# B&R Automation Studio project CarWashSimu
Automation Studio 4.12.4.107 SP; technology packages: mapp 5.23.1, mappView 5.23.0

## Configuration Config1

CPU X20CP0484-1, AutomationRuntime B4.91, Build 4.1.2, Vc V4.72.9

### Task classes (Cpu.sw)
```
Cyclic#1 (cycle 2000 us, tolerance 2000 us):
  ComTCP_P <- Libraries.ComTCP.ComTCP_P.prg
  MainCtrl <- Source.MainCtrl.MainCtrl.prg
  EntryCtrl <- Source.Entrance.EntryCtrl.prg
  ChemCtrl <- Source.Chemicals.ChemCtrl.prg
  HPWater <- Source.HPWater.HPWater.prg
  HBrushCtrl <- Source.HBrush.HBrushCtrl.prg
  VBrushCtrl <- Source.VBrush.VBrushCtrl.prg
  UBCtrl <- Source.OptUnderBody.UBCtrl.prg
  HPolish <- Source.HPolishp.HPolish.prg
  VPolishCtr <- Source.OptVpolish.VPolishCtr.prg
  WaxCtrl <- Source.OptWax.WaxCtrl.prg
  DryHCtrl <- Source.Drying.DryHCtrl.prg
  DryH2Ctrl <- Source.Drying.DryH2Ctrl.prg
  CarExit <- Source.CarExit.CarExit.prg
  Auxillary <- Source.Auxillary.Auxillary.prg
Cyclic#3 (cycle 50000 us, tolerance 50000 us):
  AlarmCtrl <- Source.Infrastructure.AlarmCtrl.AlarmCtrl.prg
  RecipeCtrl <- Source.Infrastructure.RecipeCtrl.RecipeCtrl.prg
  DataCtrl <- Source.Infrastructure.DataCtrl.DataCtrl.prg
Cyclic#4 (cycle 100000 us, tolerance 100000 us):
  Dist <- Source.Dist.prg
Cyclic#5 (cycle 200000 us, tolerance 200000 us):
  VisuCtrl <- Source.VisuCtrl.VisuCtrl.prg
Binaries: FWRules, mvLoader, TCData, udbdef, iomap, asfw, Role, sysconf, arconfig, ashwd, User, ashwac
Libraries: ComTCP_L, AsTCP, operator, runtime, astime, standard, ArEventLog, AsBrStr, MpAlarmX, MpBase, MpData, FileIO, DataObj, sys_lib, brsystem, sys_lib, arssl, fileio, asieccon, brsystem, loopconr
```

### Hardware
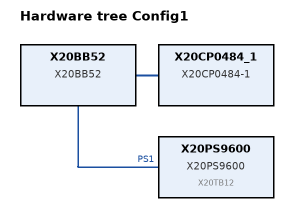
```
X20BB52 : X20BB52 v1.2.0.0
X20CP0484_1 : X20CP0484-1 v1.4.0.0  [SL -> X20BB52.SL1]
  Connector IF2:
    ActivateDevice = 1
  ConfigurationID = CarWashSimu_Config1
  Simulation = 1
  TimerDeviceType = SWIOTIMER
  Cyclic1Duration = 2000
  Cyclic1Tolerance = 2000
  Cyclic2Duration = 20000
  Cyclic2Tolerance = 20000
  Cyclic3Duration = 50000
  Cyclic3Tolerance = 50000
  Cyclic4Duration = 100000
  Cyclic4Tolerance = 100000
  Cyclic5Duration = 200000
  Cyclic5Tolerance = 200000
  Cyclic6Duration = 500000
  Cyclic6Tolerance = 500000
  Cyclic7Duration = 1000000
  Cyclic7Tolerance = 1000000
  Cyclic8Duration = 10000
  Cyclic8Tolerance = 30000000
  FileDevice1
  FileDeviceName1 = USER
  FileDevicePath1 = USER_PATH
X20PS9600 : X20PS9600 v1.6.0.0  [PS -> X20BB52.PS1; SS1 -> X20TB12.SS]
X20TB12 : X20TB12 v1.0.0.0
```

### PvMap.vvm - X20CP0484_1/PvMap.vvm
```iecst
VAR_CONFIG
	::ChemCtrl:iChem.IO.doChemRefill AT %Q.::ComTCP_SimOutputs.doChemRefill; (*Insert your comment here...*)
	::VPolishCtr:iVPolish.IO.aoVPLVel AT %Q.::ComTCP_SimOutputs.aoVPolishLVel; (*Insert your comment here...*)
	::VPolishCtr:iVPolish.IO.aoVPRVel AT %Q.::ComTCP_SimOutputs.aoVPolishRVel; (*Insert your comment here...*)
	::VPolishCtr:iVPolish.IO.doRelayRClose AT %Q.::ComTCP_SimOutputs.doVPolishRelayRClose; (*Insert your comment here...*)
	::VPolishCtr:iVPolish.IO.doRelayLClose AT %Q.::ComTCP_SimOutputs.doVPolishRelayLClose; (*Insert your comment here...*)
	::VPolishCtr:iVPolish.IO.doRelayLOpen AT %Q.::ComTCP_SimOutputs.doVPolishRelayLOpen; (*Insert your comment here...*)
	::VPolishCtr:iVPolish.IO.doRelayBrush AT %Q.::ComTCP_SimOutputs.doVPolishRelayBrush; (*Insert your comment here...*)
	::VPolishCtr:iVPolish.IO.doRelayROpen AT %Q.::ComTCP_SimOutputs.doVPolishRelayROpen; (*Insert your comment here...*)
	::ComTCP_SimInputs.aiVPolishRForceS AT %Q.::VPolishCtr:iVPolish.IO.aiVPRForceS; (*Insert your comment here...*)
	::ComTCP_SimInputs.aiVPolishRForceF AT %Q.::VPolishCtr:iVPolish.IO.aiVPRForceF; (*Insert your comment here...*)
	::ComTCP_SimInputs.aiVPolishLForceS AT %Q.::VPolishCtr:iVPolish.IO.aiVPLForceS; (*Insert your comment here...*)
	::ComTCP_SimInputs.aiVPolishLForceF AT %Q.::VPolishCtr:iVPolish.IO.aiVPLForceF; (*Insert your comment here...*)
	::CarExit:iExit.IO.doOrangeLight AT %Q.::ComTCP_SimOutputs.doExitOrangeLight; (*Insert your comment here...*)
	::CarExit:iExit.IO.doRedLight AT %Q.::ComTCP_SimOutputs.doExitRedLight; (*Insert your comment here...*)
	::ComTCP_SimOutputs.doExitGreenLight AT %Q.::ComTCP_SimOutputs.doExitGreenLight; (*Insert your comment here...*)
	::ComTCP_SimOutputs.doExitLiftDoorRelay AT %Q.::CarExit:iExit.IO.doRelayLiftDoor; (*Insert your comment here...*)
	::CarExit:iExit.IO.doRelayLowerdDoor AT %Q.::ComTCP_SimOutputs.doExitLowerDoorRelay; (*Insert your comment here...*)
	::MainCtrl:ScalDirt.y AT %Q.::ChemCtrl:iChem.IO.aoChemChemValve; (*Insert your comment here...*)
	::VBrushCtrl:iVBrush.Par.LeftVel AT %Q.::ComTCP_SimOutputs.aoVBrushLVel; (*Insert your comment here...*)
	::VBrushCtrl:iVBrush.Par.RightVel AT %Q.::ComTCP_SimOutputs.aoVBrushRVel; (*Insert your comment here...*)
	::Auxillary:iAuxillary.doRelayConv AT %Q.::ComTCP_SimOutputs.doConvRelay; (*Insert your comment here...*)
	::ChemCtrl:iChem.IO.doChemWaterValve AT %Q.::ComTCP_SimOutputs.doChemWaterValve; (*Insert your comment here...*)
	::ComTCP_SimInputs.aiEntranceSoilLevel AT %Q.::EntryCtrl:iEntry.IO.diSensSoilLvl; (*Insert your comment here...*)
	::ComTCP_SimInputs.aiVBrushLForceF AT %Q.::VBrushCtrl:iVBrush.IO.aiVBLForceF; (*Insert your comment here...*)
	::ComTCP_SimInputs.aiVBrushLForceS AT %Q.::VBrushCtrl:iVBrush.IO.aiVBLForceS; (*Insert your comment here...*)
	::ComTCP_SimInputs.aiVBrushRForceF AT %Q.::VBrushCtrl:iVBrush.IO.aiVBRForceF; (*Insert your comment here...*)
	::ComTCP_SimInputs.aiVBrushRForceS AT %Q.::VBrushCtrl:iVBrush.IO.aiVBRForceS; (*Insert your comment here...*)
	::ComTCP_SimInputs.diEmergencyStop AT %Q.::gMain.Cmd.EStop; (*Insert your comment here...*)
	::ComTCP_SimInputs.diEntranceSensor AT %Q.::EntryCtrl:iEntry.IO.diSensEntry; (*Insert your comment here...*)
	::ComTCP_SimInputs.diHBrushSensor1 AT %Q.::HBrushCtrl:iHBrush.IO.diSensHB1; (*Insert your comment here...*)
	::ComTCP_SimInputs.diHBrushSensor2 AT %Q.::HBrushCtrl:iHBrush.IO.diSensHB2; (*Insert your comment here...*)
	::ComTCP_SimInputs.diHBrushSensor3 AT %Q.::HBrushCtrl:iHBrush.IO.diSensHB3; (*Insert your comment here...*)
	::ComTCP_SimInputs.diHBrushSensor4 AT %Q.::HBrushCtrl:iHBrush.IO.diSensHB4; (*Insert your comment here...*)
	::ComTCP_SimInputs.diHighPressSensor1 AT %Q.::HPWater:iHighPress.IO.diSensHP1; (*Insert your comment here...*)
	::ComTCP_SimInputs.diHighPressSensor2 AT %Q.::HPWater:iHighPress.IO.diSensHP2; (*Insert your comment here...*)
	::ComTCP_SimInputs.diHighPressSensor3 AT %Q.::HPWater:iHighPress.IO.diSensHP3; (*Insert your comment here...*)
	::ComTCP_SimInputs.diHighPressSensor4 AT %Q.::HPWater:iHighPress.IO.diSensHP4; (*Insert your comment here...*)
	::ComTCP_SimInputs.diHPolishSensor1 AT %Q.::HPolish:iHPolish.IO.diSensHPolish1; (*Insert your comment here...*)
	::ComTCP_SimInputs.diHPolishSensor2 AT %Q.::HPolish:iHPolish.IO.diSensHPolish2; (*Insert your comment here...*)
	::ComTCP_SimInputs.diHPolishSensor3 AT %Q.::HPolish:iHPolish.IO.diSensHPolish3; (*Insert your comment here...*)
	::ComTCP_SimInputs.diHPolishSensor4 AT %Q.::HPolish:iHPolish.IO.diSensHPolish4; (*Insert your comment here...*)
	::HBrushCtrl:iHBrush.IO.doRelayHBBrush AT %Q.::ComTCP_SimOutputs.doHBrushBrushRelay; (*Insert your comment here...*)
	::HBrushCtrl:iHBrush.IO.doRelayHBLift AT %Q.::ComTCP_SimOutputs.doHBrushLiftRelay; (*Insert your comment here...*)
	::HBrushCtrl:iHBrush.IO.doRelayHBLower AT %Q.::ComTCP_SimOutputs.doHBrushLowerRelay; (*Insert your comment here...*)
	::HBrushCtrl:iHBrush.IO.doValveHB AT %Q.::ComTCP_SimOutputs.doHBrushValve; (*Insert your comment here...*)
	::HPolish:iHPolish.IO.doRelayBrush AT %Q.::ComTCP_SimOutputs.doHPolishBrushRelay; (*Insert your comment here...*)
	::HPolish:iHPolish.IO.doRelayLift AT %Q.::ComTCP_SimOutputs.doHPolishLiftRelay; (*Insert your comment here...*)
	::HPolish:iHPolish.IO.doRelayLower AT %Q.::ComTCP_SimOutputs.doHPolishLowerRelay; (*Insert your comment here...*)
	::HPWater:iHighPress.IO.doRelayHPLift AT %Q.::ComTCP_SimOutputs.doHighPressLiftRelay; (*Insert your comment here...*)
	::HPWater:iHighPress.IO.doRelayHPLow AT %Q.::ComTCP_SimOutputs.doHighPressLowerRelay; (*Insert your comment here...*)
	::HPWater:iHighPress.IO.doRelayHPPump AT %Q.::ComTCP_SimOutputs.doHighPressPumpRelay; (*Insert your comment here...*)
	::HPWater:iHighPress.IO.doValveHP AT %Q.::ComTCP_SimOutputs.doHighPressValve; (*Insert your comment here...*)
	::UBCtrl:iUBody.IO.doRelayPump AT %Q.::ComTCP_SimOutputs.doUnderbodyPumpRelay; (*Insert your comment here...*)
	::UBCtrl:iUBody.IO.doValveUB AT %Q.::ComTCP_SimOutputs.doUnderbodyValve; (*Insert your comment here...*)
	::VBrushCtrl:iVBrush.IO.doRelayVBLClose AT %Q.::ComTCP_SimOutputs.doVBrushRelayLClose; (*Insert your comment here...*)
	::VBrushCtrl:iVBrush.IO.doRelayVBLOpen AT %Q.::ComTCP_SimOutputs.doVBrushRelayLOpen; (*Insert your comment here...*)
	::VBrushCtrl:iVBrush.IO.doRelayVBRClose AT %Q.::ComTCP_SimOutputs.doVBrushRelayRClose; (*Insert your comment here...*)
	::VBrushCtrl:iVBrush.IO.doRelayVBROpen AT %Q.::ComTCP_SimOutputs.doVBrushRelayROpen; (*Insert your comment here...*)
	::ComTCP_SimInputs.diHDry1Sensor1 AT %Q.::DryHCtrl:iDry.IO.diSens1Dry1; (*Insert your comment here...*)
	::ComTCP_SimInputs.diHDry1Sensor2 AT %Q.::DryHCtrl:iDry.IO.diSens1Dry2; (*Insert your comment here...*)
	::ComTCP_SimInputs.diHDry1Sensor3 AT %Q.::DryHCtrl:iDry.IO.diSens1Dry3; (*Insert your comment here...*)
	::ComTCP_SimInputs.diHDry1Sensor4 AT %Q.::DryHCtrl:iDry.IO.diSens1Dry4; (*Insert your comment here...*)
	::ComTCP_SimInputs.diHDry2Sensor1 AT %Q.::DryH2Ctrl:iDry2.IO.diSens2Dry1; (*Insert your comment here...*)
	::ComTCP_SimInputs.diHDry2Sensor2 AT %Q.::DryH2Ctrl:iDry2.IO.diSens2Dry2; (*Insert your comment here...*)
	::ComTCP_SimInputs.diHDry2Sensor3 AT %Q.::DryH2Ctrl:iDry2.IO.diSens2Dry3; (*Insert your comment here...*)
	::ComTCP_SimInputs.diHDry2Sensor4 AT %Q.::DryH2Ctrl:iDry2.IO.diSens2Dry4; (*Insert your comment here...*)
	::DryHCtrl:iDry.IO.doRelayHD1Vent AT %Q.::ComTCP_SimOutputs.doHDry1VentRelay; (*Insert your comment here...*)
	::DryHCtrl:iDry.IO.doRelayHD1Heater AT %Q.::ComTCP_SimOutputs.doHDry1HeaterRelay; (*Insert your comment here...*)
	::DryHCtrl:iDry.IO.doRelayHD1Lower AT %Q.::ComTCP_SimOutputs.doHDry1LowerRelay; (*Insert your comment here...*)
	::DryHCtrl:iDry.IO.doRelayHD1Lift AT %Q.::ComTCP_SimOutputs.doHDry1LiftRelay; (*Insert your comment here...*)
	::DryH2Ctrl:iDry2.IO.doRelayHD2Vent AT %Q.::ComTCP_SimOutputs.doHDry2VentRelay; (*Insert your comment here...*)
	::DryH2Ctrl:iDry2.IO.doRelayHD2Heater AT %Q.::ComTCP_SimOutputs.doHDry2HeaterRelay; (*Insert your comment here...*)
	::DryH2Ctrl:iDry2.IO.doRelayHD2Lower AT %Q.::ComTCP_SimOutputs.doHDry2LowerRelay; (*Insert your comment here...*)
	::DryHCtrl:iDry.IO.doRelayVDHeater AT %Q.::ComTCP_SimOutputs.doVDry1HeaterRelay; (*Insert your comment here...*)
	::DryHCtrl:iDry.IO.doRelayVDVent AT %Q.::ComTCP_SimOutputs.doVDry1VentRelay; (*Insert your comment here...*)
	::DryH2Ctrl:iDry2.IO.doRelayHD2Lift AT %Q.::ComTCP_SimOutputs.doHDry2LiftRelay; (*Insert your comment here...*)
	::WaxCtrl:iWax.IO.doValveWax AT %Q.::ComTCP_SimOutputs.doWaxValve; (*Insert your comment here...*)
	::WaxCtrl:iWax.IO.doRefillWax AT %Q.::ComTCP_SimOutputs.doWaxRefill; (*Insert your comment here...*)
	::WaxCtrl:iWax.IO.doRealyWaxPump AT %Q.::ComTCP_SimOutputs.doWaxPumpRelay; (*Insert your comment here...*)
END_VAR
```

### Config.mpalarmxcore - X20CP0484_1/mappServices/Config.mpalarmxcore
```
Element gAlarmXCore (Type=mpalarmxcore)
  mapp.AlarmX.Core:
    BySeverity:
      [0]:
        Severity = 100
        [0] = Reaction
          Name = EStopErr
  mapp.AlarmX.Core.Configuration:
    [0]:
      Name = EStopChem
      Message = EStop Pressed chemical control
      Severity = 100
      Behavior = PersistentAlarm
    [1]:
      Name = EStopHighPre
      Message = EStop Pressed High pressurecontrol
      Severity = 100
      Behavior = PersistentAlarm
    [2]:
      Name = EStopHB
      Message = EStop Pressed horizontal brush control
      Severity = 100
      Behavior = PersistentAlarm
    [3]:
      Name = EStopVB
      Message = EStop Pressed vertical brush control
      Severity = 100
      Behavior = PersistentAlarm
    [4]:
      Name = EStopUB
      Message = EStop Pressed under body control
      Severity = 100
      Behavior = PersistentAlarm
    [5]:
      Name = EStopVPol
      Message = Estop Pressed Vertical polish
      Severity = 100
      Behavior = PersistentAlarm
    [6]:
      Name = EStopDry
      Message = EStop Pressed Dry control
      Severity = 100
      Behavior = PersistentAlarm
    [7]:
      Name = EStopHWax
      Message = EStop Pressed HotWax control
      Severity = 100
      Behavior = PersistentAlarm
    [8]:
      Name = EStopConv
      Message = EStop Pressed Conveyor control
      Severity = 100
      Behavior = PersistentAlarm
    [9]:
      Name = WaterLow
      Message = Water level is low
      Severity = 100
      Behavior = PersistentAlarm
    [10]:
      Name = ChemLow
      Message = Chemical level is low
      Severity = 50
      Behavior = PersistentAlarm
    [11]:
      Name = WaxLow
      Message = Wax level is low
      Severity = 50
      Behavior = PersistentAlarm
    [12]:
      Name = EStopEntry
      Message = Emergency stop of entry is pressed
      Severity = 100
      Behavior = PersistentAlarm
    [13]:
      Name = EStopHPol
      Message = Estop Pressed Horizonatal polish
      Severity = 100
      Behavior = PersistentAlarm
    [14]:
      Name = EStopExit
      Message = EStop of exit is pressed
      Severity = 100
      Behavior = PersistentAlarm
Element gAlarmXCore_1 (Type=mpalarmxcore)
```

## Logical view

Binary libraries used (declarations not repeated): operator, runtime, astime, AsIecCon, AsTCP, standard, ArEventLog, AsBrStr, LoopConR, sys_lib, brsystem, MpAlarmX, MpBase, MpData, FileIO, DataObj

### Global.typ - Global data types
```iecst
TYPE
	MainCmd_typ : 	STRUCT
		Start : BOOL;
		Stop : BOOL;
		EStop : BOOL;
	END_STRUCT;
	MainOption_typ : 	STRUCT
		EntryState : BOOL;
		ChemicalState : BOOL;
		HighPress : BOOL;
		HBrush : BOOL;
		Polish : BOOL;
		UnderBody : BOOL;
		Wax : BOOL;
		VBrush : BOOL;
		Dry : BOOL;
	END_STRUCT;
	MainCtrl_typ : 	STRUCT
		Cmd : MainCmd_typ;
		Option : MainOption_typ;
	END_STRUCT;
END_TYPE
```

### Global.var - Global variables
```iecst
VAR
	gMi_Mode2 : BOOL;
	gMi_Mode3 : BOOL;
	gMi_Mode4 : BOOL;
	gMi_Mode1 : BOOL;
	gMain : MainCtrl_typ;
	iVa_Distance : REAL;
	gCar : ARRAY[0..2] OF BOOL;
END_VAR
```

### Package Logical/Libraries - Global libraries

### Library Logical/Libraries/ComTCP/ComTCP_L (ANSIC)
Depends on: AsTCP, operator, runtime, astime, standard, ArEventLog, AsBrStr

#### MNG_Global.hpp
```cpp
#ifndef  _MNGGLOBAL_HPP_
#define _MNGGLOBAL_HPP_

#include <mng_globalTYP.h>

    typedef struct {

		signed short NumSignals;

        /* BOOL diEmergencyStop */
        BOOL diEmergencyStop;
        /* BOOL diEntranceSensor */
        BOOL diEntranceSensor;
        /* REAL aiEntranceSoilLevel */
        REAL aiEntranceSoilLevel;
        /* BOOL diHighPressSensor1 */
        BOOL diHighPressSensor1;
        /* BOOL diHighPressSensor2 */
        BOOL diHighPressSensor2;
        /* BOOL diHighPressSensor3 */
        BOOL diHighPressSensor3;
        /* BOOL diHighPressSensor4 */
        BOOL diHighPressSensor4;
        /* BOOL diHBrushSensor1 */
        BOOL diHBrushSensor1;
        /* BOOL diHBrushSensor2 */
        BOOL diHBrushSensor2;
        /* BOOL diHBrushSensor3 */
        BOOL diHBrushSensor3;
        /* BOOL diHBrushSensor4 */
        BOOL diHBrushSensor4;
        /* REAL aiVBrushLForceF */
        REAL aiVBrushLForceF;
        /* REAL aiVBrushLForceS */
        REAL aiVBrushLForceS;
        /* REAL aiVBrushRForceF */
        REAL aiVBrushRForceF;
        /* REAL aiVBrushRForceS */
        REAL aiVBrushRForceS;
        /* BOOL diHPolishSensor1 */
        BOOL diHPolishSensor1;
        /* BOOL diHPolishSensor2 */
        BOOL diHPolishSensor2;
        /* BOOL diHPolishSensor3 */
        BOOL diHPolishSensor3;
        /* BOOL diHPolishSensor4 */
        BOOL diHPolishSensor4;
        /* REAL aiVPolishLForceF */
        REAL aiVPolishLForceF;
        /* REAL aiVPolishLForceS */
        REAL aiVPolishLForceS;
        /* REAL aiVPolishRForceF */
        REAL aiVPolishRForceF;
        /* REAL aiVPolishRForceS */
        REAL aiVPolishRForceS;
        /* BOOL diHDry1Sensor1 */
        BOOL diHDry1Sensor1;
        /* BOOL diHDry1Sensor2 */
        BOOL diHDry1Sensor2;
        /* BOOL diHDry1Sensor3 */
        BOOL diHDry1Sensor3;
        /* BOOL diHDry1Sensor4 */
        BOOL diHDry1Sensor4;
        /* BOOL diHDry2Sensor1 */
        BOOL diHDry2Sensor1;
        /* BOOL diHDry2Sensor2 */
        BOOL diHDry2Sensor2;
        /* BOOL diHDry2Sensor3 */
        BOOL diHDry2Sensor3;
        /* BOOL diHDry2Sensor4 */
        BOOL diHDry2Sensor4;
        /* REAL aiWaterLevel */
        REAL aiWaterLevel;

        } ComTCP_INPUTS_32BIT_FWRD;

    typedef struct {

		signed short NumSignals;

        /* BOOL doMaintenanceMode */
        BOOL doMaintenanceMode;
        /* REAL aoChemChemValve */
        REAL aoChemChemValve;
        /* BOOL doChemWaterValve */
        BOOL doChemWaterValve;
        /* BOOL doChemRefill */
        BOOL doChemRefill;
        /* BOOL doHighPressLiftRelay */
        BOOL doHighPressLiftRelay;
        /* BOOL doHighPressLowerRelay */
        BOOL doHighPressLowerRelay;
        /* BOOL doHighPressValve */
        BOOL doHighPressValve;
        /* BOOL doHighPressPumpRelay */
        BOOL doHighPressPumpRelay;
        /* BOOL doHBrushLiftRelay */
        BOOL doHBrushLiftRelay;
        /* BOOL doHBrushLowerRelay */
        BOOL doHBrushLowerRelay;
        /* BOOL doHBrushValve */
        BOOL doHBrushValve;
        /* BOOL doHBrushBrushRelay */
        BOOL doHBrushBrushRelay;
        /* BOOL doVBrushRelayLClose */
        BOOL doVBrushRelayLClose;
        /* BOOL doVBrushRelayLOpen */
        BOOL doVBrushRelayLOpen;
        /* BOOL doVBrushRelayRClose */
        BOOL doVBrushRelayRClose;
        /* BOOL doVBrushRelayROpen */
        BOOL doVBrushRelayROpen;
        /* REAL aoVBrushLVel */
        REAL aoVBrushLVel;
        /* REAL aoVBrushRVel */
        REAL aoVBrushRVel;
        /* BOOL doVBrushValve */
        BOOL doVBrushValve;
        /* BOOL doVBrushRelayBrush */
        BOOL doVBrushRelayBrush;
        /* BOOL doUnderbodyValve */
        BOOL doUnderbodyValve;
        /* BOOL doUnderbodyPumpRelay */
        BOOL doUnderbodyPumpRelay;
        /* BOOL doHPolishLiftRelay */
        BOOL doHPolishLiftRelay;
        /* BOOL doHPolishLowerRelay */
        BOOL doHPolishLowerRelay;
        /* BOOL doHPolishBrushRelay */
        BOOL doHPolishBrushRelay;
        /* BOOL doVPolishRelayLClose */
        BOOL doVPolishRelayLClose;
        /* BOOL doVPolishRelayLOpen */
        BOOL doVPolishRelayLOpen;
        /* BOOL doVPolishRelayRClose */
        BOOL doVPolishRelayRClose;
        /* BOOL doVPolishRelayROpen */
        BOOL doVPolishRelayROpen;
        /* REAL aoVPolishLVel */
        REAL aoVPolishLVel;
        /* REAL aoVPolishRVel */
        REAL aoVPolishRVel;
        /* BOOL doVPolishRelayBrush */
        BOOL doVPolishRelayBrush;
        /* BOOL doWaxValve */
        BOOL doWaxValve;
        /* BOOL doWaxPumpRelay */
        BOOL doWaxPumpRelay;
        /* BOOL doWaxRefill */
        BOOL doWaxRefill;
        /* BOOL doHDry1LiftRelay */
        BOOL doHDry1LiftRelay;
        /* BOOL doHDry1LowerRelay */
        BOOL doHDry1LowerRelay;
        /* BOOL doHDry1VentRelay */
        BOOL doHDry1VentRelay;
        /* BOOL doHDry1HeaterRelay */
        BOOL doHDry1HeaterRelay;
        /* BOOL doVDry1VentRelay */
        BOOL doVDry1VentRelay;
        /* BOOL doVDry1HeaterRelay */
        BOOL doVDry1HeaterRelay;
        /* BOOL doHDry2LiftRelay */
        BOOL doHDry2LiftRelay;
        /* BOOL doHDry2LowerRelay */
        BOOL doHDry2LowerRelay;
        /* BOOL doHDry2VentRelay */
        BOOL doHDry2VentRelay;
        /* BOOL doHDry2HeaterRelay */
        BOOL doHDry2HeaterRelay;
        /* BOOL doConvRelay */
        BOOL doConvRelay;
        /* BOOL doWaterValve */
        BOOL doWaterValve;
        /* BOOL doTankWaterValve */
        BOOL doTankWaterValve;
        /* BOOL doExitGreenLight */
        BOOL doExitGreenLight;
        /* BOOL doExitOrangeLight */
        BOOL doExitOrangeLight;
        /* BOOL doExitRedLight */
        BOOL doExitRedLight;
        /* BOOL doExitLiftDoorRelay */
        BOOL doExitLiftDoorRelay;
        /* BOOL doExitLowerDoorRelay */
        BOOL doExitLowerDoorRelay;

        } ComTCP_OUTPUTS_32BIT_FWRD;

#endif
```

#### MNG_CpyOutToMsg.cpp
```cpp
#include "MNG_InternalTyp.hpp"

unsigned long int MNG_CpyOutToMsg(MNG_RawDatagram * pToServer, unsigned long int counter, ComTCP_OUTPUTS_32BIT_FWRD *pSimOutputs ) {

        unsigned long int DWordBuffer;

        pSimOutputs->NumSignals = 53;
        (pToServer->Header).ByteCount    = H_TO_NUDINT(216);
        (pToServer->Header).DatagramType = H_TO_NUDINT(MNG_Raw32BitImage);
        (pToServer->Header).SentTime = H_TO_NUDINT(0);  // Todo
        (pToServer->Header).Counter = H_TO_NUDINT(counter);
        pToServer->Payload[0] = H_TO_NUDINT(pSimOutputs->NumSignals);

    /* doMaintenanceMode : BOOL */
    if(pSimOutputs->doMaintenanceMode == 1) {
        pToServer->Payload[1] = 0xFFFFFFFF;   /*BOOL */
    } else {
        pToServer->Payload[1] = 0;
    }

    /* aoChemChemValve : FLOAT32 */
    brsmemcpy((unsigned long int)&(DWordBuffer), (unsigned long int)&(pSimOutputs->aoChemChemValve), 4);
    pToServer->Payload[2] = H_TO_NUDINT(DWordBuffer);

    /* doChemWaterValve : BOOL */
    if(pSimOutputs->doChemWaterValve == 1) {
        pToServer->Payload[3] = 0xFFFFFFFF;   /*BOOL */
    } else {
        pToServer->Payload[3] = 0;
    }

    /* doChemRefill : BOOL */
    if(pSimOutputs->doChemRefill == 1) {
        pToServer->Payload[4] = 0xFFFFFFFF;   /*BOOL */
    } else {
        pToServer->Payload[4] = 0;
    }

    /* doHighPressLiftRelay : BOOL */
    if(pSimOutputs->doHighPressLiftRelay == 1) {
        pToServer->Payload[5] = 0xFFFFFFFF;   /*BOOL */
    } else {
        pToServer->Payload[5] = 0;
    }

    /* doHighPressLowerRelay : BOOL */
    if(pSimOutputs->doHighPressLowerRelay == 1) {
        pToServer->Payload[6] = 0xFFFFFFFF;   /*BOOL */
    } else {
        pToServer->Payload[6] = 0;
    }

    /* doHighPressValve : BOOL */
    if(pSimOutputs->doHighPressValve == 1) {
        pToServer->Payload[7] = 0xFFFFFFFF;   /*BOOL */
    } else {
        pToServer->Payload[7] = 0;
    }

    /* doHighPressPumpRelay : BOOL */
    if(pSimOutputs->doHighPressPumpRelay == 1) {
        pToServer->Payload[8] = 0xFFFFFFFF;   /*BOOL */
    } else {
        pToServer->Payload[8] = 0;
    }

    /* doHBrushLiftRelay : BOOL */
    if(pSimOutputs->doHBrushLiftRelay == 1) {
        pToServer->Payload[9] = 0xFFFFFFFF;   /*BOOL */
    } else {
        pToServer->Payload[9] = 0;
    }

    /* doHBrushLowerRelay : BOOL */
    if(pSimOutputs->doHBrushLowerRelay == 1) {
        pToServer->Payload[10] = 0xFFFFFFFF;   /*BOOL */
    } else {
        pToServer->Payload[10] = 0;
    }

    /* doHBrushValve : BOOL */
    if(pSimOutputs->doHBrushValve == 1) {
        pToServer->Payload[11] = 0xFFFFFFFF;   /*BOOL */
    } else {
        pToServer->Payload[11] = 0;
    }

    /* doHBrushBrushRelay : BOOL */
    if(pSimOutputs->doHBrushBrushRelay == 1) {
        pToServer->Payload[12] = 0xFFFFFFFF;   /*BOOL */
    } else {
        pToServer->Payload[12] = 0;
    }

    /* doVBrushRelayLClose : BOOL */
    if(pSimOutputs->doVBrushRelayLClose == 1) {
        pToServer->Payload[13] = 0xFFFFFFFF;   /*BOOL */
    } else {
        pToServer->Payload[13] = 0;
    }

    /* doVBrushRelayLOpen : BOOL */
    if(pSimOutputs->doVBrushRelayLOpen == 1) {
        pToServer->Payload[14] = 0xFFFFFFFF;   /*BOOL */
    } else {
        pToServer->Payload[14] = 0;
    }

    /* doVBrushRelayRClose : BOOL */
    if(pSimOutputs->doVBrushRelayRClose == 1) {
        pToServer->Payload[15] = 0xFFFFFFFF;   /*BOOL */
    } else {
        pToServer->Payload[15] = 0;
    }

    /* doVBrushRelayROpen : BOOL */
    if(pSimOutputs->doVBrushRelayROpen == 1) {
        pToServer->Payload[16] = 0xFFFFFFFF;   /*BOOL */
    } else {
        pToServer->Payload[16] = 0;
    }

    /* aoVBrushLVel : FLOAT32 */
    brsmemcpy((unsigned long int)&(DWordBuffer), (unsigned long int)&(pSimOutputs->aoVBrushLVel), 4);
    pToServer->Payload[17] = H_TO_NUDINT(DWordBuffer);

    /* aoVBrushRVel : FLOAT32 */
    brsmemcpy((unsigned long int)&(DWordBuffer), (unsigned long int)&(pSimOutputs->aoVBrushRVel), 4);
    pToServer->Payload[18] = H_TO_NUDINT(DWordBuffer);

    /* doVBrushValve : BOOL */
    if(pSimOutputs->doVBrushValve == 1) {
        pToServer->Payload[19] = 0xFFFFFFFF;   /*BOOL */
    } else {
        pToServer->Payload[19] = 0;
    }

    /* doVBrushRelayBrush : BOOL */
    if(pSimOutputs->doVBrushRelayBrush == 1) {
        pToServer->Payload[20] = 0xFFFFFFFF;   /*BOOL */
    } else {
        pToServer->Payload[20] = 0;
    }

    /* doUnderbodyValve : BOOL */
    if(pSimOutputs->doUnderbodyValve == 1) {
        pToServer->Payload[21] = 0xFFFFFFFF;   /*BOOL */
    } else {
        pToServer->Payload[21] = 0;
    }

    /* doUnderbodyPumpRelay : BOOL */
    if(pSimOutputs->doUnderbodyPumpRelay == 1) {
        pToServer->Payload[22] = 0xFFFFFFFF;   /*BOOL */
    } else {
        pToServer->Payload[22] = 0;
    }

    /* doHPolishLiftRelay : BOOL */
    if(pSimOutputs->doHPolishLiftRelay == 1) {
        pToServer->Payload[23] = 0xFFFFFFFF;   /*BOOL */
    } else {
        pToServer->Payload[23] = 0;
    }

    /* doHPolishLowerRelay : BOOL */
    if(pSimOutputs->doHPolishLowerRelay == 1) {
        pToServer->Payload[24] = 0xFFFFFFFF;   /*BOOL */
    } else {
        pToServer->Payload[24] = 0;
    }

    /* doHPolishBrushRelay : BOOL */
    if(pSimOutputs->doHPolishBrushRelay == 1) {
        pToServer->Payload[25] = 0xFFFFFFFF;   /*BOOL */
    } else {
        pToServer->Payload[25] = 0;
    }

    /* doVPolishRelayLClose : BOOL */
    if(pSimOutputs->doVPolishRelayLClose == 1) {
        pToServer->Payload[26] = 0xFFFFFFFF;   /*BOOL */
    } else {
        pToServer->Payload[26] = 0;
    }

    /* doVPolishRelayLOpen : BOOL */
    if(pSimOutputs->doVPolishRelayLOpen == 1) {
        pToServer->Payload[27] = 0xFFFFFFFF;   /*BOOL */
    } else {
        pToServer->Payload[27] = 0;
    }

    /* doVPolishRelayRClose : BOOL */
    if(pSimOutputs->doVPolishRelayRClose == 1) {
        pToServer->Payload[28] = 0xFFFFFFFF;   /*BOOL */
    } else {
        pToServer->Payload[28] = 0;
    }

    /* doVPolishRelayROpen : BOOL */
    if(pSimOutputs->doVPolishRelayROpen == 1) {
        pToServer->Payload[29] = 0xFFFFFFFF;   /*BOOL */
    } else {
        pToServer->Payload[29] = 0;
    }

    /* aoVPolishLVel : FLOAT32 */
    brsmemcpy((unsigned long int)&(DWordBuffer), (unsigned long int)&(pSimOutputs->aoVPolishLVel), 4);
    pToServer->Payload[30] = H_TO_NUDINT(DWordBuffer);

    /* aoVPolishRVel : FLOAT32 */
    brsmemcpy((unsigned long int)&(DWordBuffer), (unsigned long int)&(pSimOutputs->aoVPolishRVel), 4);
    pToServer->Payload[31] = H_TO_NUDINT(DWordBuffer);

    /* doVPolishRelayBrush : BOOL */
    if(pSimOutputs->doVPolishRelayBrush == 1) {
        pToServer->Payload[32] = 0xFFFFFFFF;   /*BOOL */
    } else {
        pToServer->Payload[32] = 0;
    }

    /* doWaxValve : BOOL */
    if(pSimOutputs->doWaxValve == 1) {
        pToServer->Payload[33] = 0xFFFFFFFF;   /*BOOL */
    } else {
        pToServer->Payload[33] = 0;
    }

    /* doWaxPumpRelay : BOOL */
    if(pSimOutputs->doWaxPumpRelay == 1) {
        pToServer->Payload[34] = 0xFFFFFFFF;   /*BOOL */
    } else {
        pToServer->Payload[34] = 0;
    }

    /* doWaxRefill : BOOL */
    if(pSimOutputs->doWaxRefill == 1) {
        pToServer->Payload[35] = 0xFFFFFFFF;   /*BOOL */
    } else {
        pToServer->Payload[35] = 0;
    }

    /* doHDry1LiftRelay : BOOL */
    if(pSimOutputs->doHDry1LiftRelay == 1) {
        pToServer->Payload[36] = 0xFFFFFFFF;   /*BOOL */
    } else {
        pToServer->Payload[36] = 0;
    }

    /* doHDry1LowerRelay : BOOL */
    if(pSimOutputs->doHDry1LowerRelay == 1) {
        pToServer->Payload[37] = 0xFFFFFFFF;   /*BOOL */
    } else {
        pToServer->Payload[37] = 0;
    }

    /* doHDry1VentRelay : BOOL */
    if(pSimOutputs->doHDry1VentRelay == 1) {
        pToServer->Payload[38] = 0xFFFFFFFF;   /*BOOL */
    } else {
        pToServer->Payload[38] = 0;
    }

    /* doHDry1HeaterRelay : BOOL */
    if(pSimOutputs->doHDry1HeaterRelay == 1) {
        pToServer->Payload[39] = 0xFFFFFFFF;   /*BOOL */
    } else {
        pToServer->Payload[39] = 0;
    }

    /* doVDry1VentRelay : BOOL */
    if(pSimOutputs->doVDry1VentRelay == 1) {
        pToServer->Payload[40] = 0xFFFFFFFF;   /*BOOL */
    } else {
        pToServer->Payload[40] = 0;
    }

    /* doVDry1HeaterRelay : BOOL */
    if(pSimOutputs->doVDry1HeaterRelay == 1) {
        pToServer->Payload[41] = 0xFFFFFFFF;   /*BOOL */
    } else {
        pToServer->Payload[41] = 0;
    }

    /* doHDry2LiftRelay : BOOL */
    if(pSimOutputs->doHDry2LiftRelay == 1) {
        pToServer->Payload[42] = 0xFFFFFFFF;   /*BOOL */
    } else {
        pToServer->Payload[42] = 0;
    }

    /* doHDry2LowerRelay : BOOL */
    if(pSimOutputs->doHDry2LowerRelay == 1) {
        pToServer->Payload[43] = 0xFFFFFFFF;   /*BOOL */
    } else {
        pToServer->Payload[43] = 0;
    }

    /* doHDry2VentRelay : BOOL */
    if(pSimOutputs->doHDry2VentRelay == 1) {
        pToServer->Payload[44] = 0xFFFFFFFF;   /*BOOL */
    } else {
        pToServer->Payload[44] = 0;
    }

    /* doHDry2HeaterRelay : BOOL */
    if(pSimOutputs->doHDry2HeaterRelay == 1) {
        pToServer->Payload[45] = 0xFFFFFFFF;   /*BOOL */
    } else {
        pToServer->Payload[45] = 0;
    }

    /* doConvRelay : BOOL */
    if(pSimOutputs->doConvRelay == 1) {
        pToServer->Payload[46] = 0xFFFFFFFF;   /*BOOL */
    } else {
        pToServer->Payload[46] = 0;
    }

    /* doWaterValve : BOOL */
    if(pSimOutputs->doWaterValve == 1) {
        pToServer->Payload[47] = 0xFFFFFFFF;   /*BOOL */
    } else {
        pToServer->Payload[47] = 0;
    }

    /* doTankWaterValve : BOOL */
    if(pSimOutputs->doTankWaterValve == 1) {
        pToServer->Payload[48] = 0xFFFFFFFF;   /*BOOL */
    } else {
        pToServer->Payload[48] = 0;
    }

    /* doExitGreenLight : BOOL */
    if(pSimOutputs->doExitGreenLight == 1) {
        pToServer->Payload[49] = 0xFFFFFFFF;   /*BOOL */
    } else {
        pToServer->Payload[49] = 0;
    }

    /* doExitOrangeLight : BOOL */
    if(pSimOutputs->doExitOrangeLight == 1) {
        pToServer->Payload[50] = 0xFFFFFFFF;   /*BOOL */
    } else {
        pToServer->Payload[50] = 0;
    }

    /* doExitRedLight : BOOL */
    if(pSimOutputs->doExitRedLight == 1) {
        pToServer->Payload[51] = 0xFFFFFFFF;   /*BOOL */
    } else {
        pToServer->Payload[51] = 0;
    }

    /* doExitLiftDoorRelay : BOOL */
    if(pSimOutputs->doExitLiftDoorRelay == 1) {
        pToServer->Payload[52] = 0xFFFFFFFF;   /*BOOL */
    } else {
        pToServer->Payload[52] = 0;
    }

    /* doExitLowerDoorRelay : BOOL */
    if(pSimOutputs->doExitLowerDoorRelay == 1) {
        pToServer->Payload[53] = 0xFFFFFFFF;   /*BOOL */
    } else {
        pToServer->Payload[53] = 0;
    }

	return 0;
}
```

#### MNG_CpyMsgToInp.cpp
```cpp
#include "MNG_InternalTyp.hpp"

unsigned long int MNG_CpyMsgToInp(MNG_RawDatagram * pFromServer, ComTCP_INPUTS_32BIT_FWRD *pSimInputs) {

    MNG_DatagramType datagramType;
	unsigned long int DWordBuffer;
        unsigned long int byteCount;
	unsigned long int numSignalsInMessage;

	byteCount = N_TO_HUDINT((pFromServer->Header).ByteCount);
	datagramType = static_cast<MNG_DatagramType>(N_TO_HUDINT((pFromServer->Header).DatagramType));
	if (datagramType != MNG_Raw32BitImage) {
		return 0;
	}

    pSimInputs->NumSignals = 32;

    numSignalsInMessage = N_TO_HUDINT(pFromServer->Payload[0]);
        if ((static_cast<long int>(numSignalsInMessage) != pSimInputs->NumSignals) ||
	(byteCount != 4 + numSignalsInMessage * 4)) {
		return 0;
	}

    /* BOOL diEmergencyStop */
    pSimInputs->diEmergencyStop = (pFromServer->Payload[1] != 0);

    /* BOOL diEntranceSensor */
    pSimInputs->diEntranceSensor = (pFromServer->Payload[2] != 0);

    /* FLOAT32 aiEntranceSoilLevel */
    DWordBuffer = N_TO_HUDINT(pFromServer->Payload[3]);
    brsmemcpy((unsigned long int)&(pSimInputs->aiEntranceSoilLevel), (unsigned long int)&(DWordBuffer), 4);

    /* BOOL diHighPressSensor1 */
    pSimInputs->diHighPressSensor1 = (pFromServer->Payload[4] != 0);

    /* BOOL diHighPressSensor2 */
    pSimInputs->diHighPressSensor2 = (pFromServer->Payload[5] != 0);

    /* BOOL diHighPressSensor3 */
    pSimInputs->diHighPressSensor3 = (pFromServer->Payload[6] != 0);

    /* BOOL diHighPressSensor4 */
    pSimInputs->diHighPressSensor4 = (pFromServer->Payload[7] != 0);

    /* BOOL diHBrushSensor1 */
    pSimInputs->diHBrushSensor1 = (pFromServer->Payload[8] != 0);

    /* BOOL diHBrushSensor2 */
    pSimInputs->diHBrushSensor2 = (pFromServer->Payload[9] != 0);

    /* BOOL diHBrushSensor3 */
    pSimInputs->diHBrushSensor3 = (pFromServer->Payload[10] != 0);

    /* BOOL diHBrushSensor4 */
    pSimInputs->diHBrushSensor4 = (pFromServer->Payload[11] != 0);

    /* FLOAT32 aiVBrushLForceF */
    DWordBuffer = N_TO_HUDINT(pFromServer->Payload[12]);
    brsmemcpy((unsigned long int)&(pSimInputs->aiVBrushLForceF), (unsigned long int)&(DWordBuffer), 4);

    /* FLOAT32 aiVBrushLForceS */
    DWordBuffer = N_TO_HUDINT(pFromServer->Payload[13]);
    brsmemcpy((unsigned long int)&(pSimInputs->aiVBrushLForceS), (unsigned long int)&(DWordBuffer), 4);

    /* FLOAT32 aiVBrushRForceF */
    DWordBuffer = N_TO_HUDINT(pFromServer->Payload[14]);
    brsmemcpy((unsigned long int)&(pSimInputs->aiVBrushRForceF), (unsigned long int)&(DWordBuffer), 4);

    /* FLOAT32 aiVBrushRForceS */
    DWordBuffer = N_TO_HUDINT(pFromServer->Payload[15]);
    brsmemcpy((unsigned long int)&(pSimInputs->aiVBrushRForceS), (unsigned long int)&(DWordBuffer), 4);

    /* BOOL diHPolishSensor1 */
    pSimInputs->diHPolishSensor1 = (pFromServer->Payload[16] != 0);

    /* BOOL diHPolishSensor2 */
    pSimInputs->diHPolishSensor2 = (pFromServer->Payload[17] != 0);

    /* BOOL diHPolishSensor3 */
    pSimInputs->diHPolishSensor3 = (pFromServer->Payload[18] != 0);

    /* BOOL diHPolishSensor4 */
    pSimInputs->diHPolishSensor4 = (pFromServer->Payload[19] != 0);

    /* FLOAT32 aiVPolishLForceF */
    DWordBuffer = N_TO_HUDINT(pFromServer->Payload[20]);
    brsmemcpy((unsigned long int)&(pSimInputs->aiVPolishLForceF), (unsigned long int)&(DWordBuffer), 4);

    /* FLOAT32 aiVPolishLForceS */
    DWordBuffer = N_TO_HUDINT(pFromServer->Payload[21]);
    brsmemcpy((unsigned long int)&(pSimInputs->aiVPolishLForceS), (unsigned long int)&(DWordBuffer), 4);

    /* FLOAT32 aiVPolishRForceF */
    DWordBuffer = N_TO_HUDINT(pFromServer->Payload[22]);
    brsmemcpy((unsigned long int)&(pSimInputs->aiVPolishRForceF), (unsigned long int)&(DWordBuffer), 4);

    /* FLOAT32 aiVPolishRForceS */
    DWordBuffer = N_TO_HUDINT(pFromServer->Payload[23]);
    brsmemcpy((unsigned long int)&(pSimInputs->aiVPolishRForceS), (unsigned long int)&(DWordBuffer), 4);

    /* BOOL diHDry1Sensor1 */
    pSimInputs->diHDry1Sensor1 = (pFromServer->Payload[24] != 0);

    /* BOOL diHDry1Sensor2 */
    pSimInputs->diHDry1Sensor2 = (pFromServer->Payload[25] != 0);

    /* BOOL diHDry1Sensor3 */
    pSimInputs->diHDry1Sensor3 = (pFromServer->Payload[26] != 0);

    /* BOOL diHDry1Sensor4 */
    pSimInputs->diHDry1Sensor4 = (pFromServer->Payload[27] != 0);

    /* BOOL diHDry2Sensor1 */
    pSimInputs->diHDry2Sensor1 = (pFromServer->Payload[28] != 0);

    /* BOOL diHDry2Sensor2 */
    pSimInputs->diHDry2Sensor2 = (pFromServer->Payload[29] != 0);

    /* BOOL diHDry2Sensor3 */
    pSimInputs->diHDry2Sensor3 = (pFromServer->Payload[30] != 0);

    /* BOOL diHDry2Sensor4 */
    pSimInputs->diHDry2Sensor4 = (pFromServer->Payload[31] != 0);

    /* FLOAT32 aiWaterLevel */
    DWordBuffer = N_TO_HUDINT(pFromServer->Payload[32]);
    brsmemcpy((unsigned long int)&(pSimInputs->aiWaterLevel), (unsigned long int)&(DWordBuffer), 4);

return N_TO_HUDINT((pFromServer->Header).Counter); // return counter
}
```

### Program Logical/Libraries/ComTCP/ComTCP_P (ANSIC)

#### Main.cpp
```cpp
#include <bur/plctypes.h>

#include "../ComTCP_L/MNG_Global.hpp"
#include "../ComTCP_L/MNG_InternalTyp.hpp"
#include "../ComTCP_L/MNG_ComHdlr.hpp"

#include <MNG_PackageTyp.h>
#include <MNG_PackageVAR.h>
#include <TypesTYP.h>
#include <VariablesVAR.h>

unsigned long bur_heap_size = 0x4FFFF;

MNG_ComHdlr *pMNG_ComHdlr;

void _INIT ProgramInit(void)
{
    pMNG_ComHdlr = new MNG_ComHdlr(ComTCP_SimServerAddress, ComTCP_SimServerPort, ComTCP_SimSendCycleTime);
}

void _CYCLIC ProgramCyclic(void)
{
    connectionState = pMNG_ComHdlr->RunCommunication((void*)&ComTCP_SimInputs,(void*)&ComTCP_SimOutputs, &ComTCP_SimActive);
}

void _EXIT ProgramExit(void)
{
    delete pMNG_ComHdlr;
}
```

### MNG_Package.typ
```iecst
(*                                                                            *)
(* File generated by the B&R AS 4 control config generator                    *)
(*                                                                            *)
(*     Provider: machineering                                                 *)
(*  Application: iPhysics_2.4.master                                          *)
(* Architecture: Windows 64 Bit                                               *)
(*      Version: 2.4.12706.master                                             *)
(*        Build: 608a88cb4                                                    *)
(*         Date: 2022-08-25, Time: 10:57:22                                   *)
(*                                                                            *)

TYPE
ComTCP_INPUTS_32BIT : STRUCT

		NumSignals	: INT := 32;

        diEmergencyStop : BOOL := 0;
        (* BOOL diEmergencyStop *)
        diEntranceSensor : BOOL := 0;
        (* BOOL diEntranceSensor *)
        aiEntranceSoilLevel : REAL := 0.0;
        (* REAL aiEntranceSoilLevel *)
        diHighPressSensor1 : BOOL := 0;
        (* BOOL diHighPressSensor1 *)
        diHighPressSensor2 : BOOL := 0;
        (* BOOL diHighPressSensor2 *)
        diHighPressSensor3 : BOOL := 0;
        (* BOOL diHighPressSensor3 *)
        diHighPressSensor4 : BOOL := 0;
        (* BOOL diHighPressSensor4 *)
        diHBrushSensor1 : BOOL := 0;
        (* BOOL diHBrushSensor1 *)
        diHBrushSensor2 : BOOL := 0;
        (* BOOL diHBrushSensor2 *)
        diHBrushSensor3 : BOOL := 0;
        (* BOOL diHBrushSensor3 *)
        diHBrushSensor4 : BOOL := 0;
        (* BOOL diHBrushSensor4 *)
        aiVBrushLForceF : REAL := 0.0;
        (* REAL aiVBrushLForceF *)
        aiVBrushLForceS : REAL := 0.0;
        (* REAL aiVBrushLForceS *)
        aiVBrushRForceF : REAL := 0.0;
        (* REAL aiVBrushRForceF *)
        aiVBrushRForceS : REAL := 0.0;
        (* REAL aiVBrushRForceS *)
        diHPolishSensor1 : BOOL := 0;
        (* BOOL diHPolishSensor1 *)
        diHPolishSensor2 : BOOL := 0;
        (* BOOL diHPolishSensor2 *)
        diHPolishSensor3 : BOOL := 0;
        (* BOOL diHPolishSensor3 *)
        diHPolishSensor4 : BOOL := 0;
        (* BOOL diHPolishSensor4 *)
        aiVPolishLForceF : REAL := 0.0;
        (* REAL aiVPolishLForceF *)
        aiVPolishLForceS : REAL := 0.0;
        (* REAL aiVPolishLForceS *)
        aiVPolishRForceF : REAL := 0.0;
        (* REAL aiVPolishRForceF *)
        aiVPolishRForceS : REAL := 0.0;
        (* REAL aiVPolishRForceS *)
        diHDry1Sensor1 : BOOL := 0;
        (* BOOL diHDry1Sensor1 *)
        diHDry1Sensor2 : BOOL := 0;
        (* BOOL diHDry1Sensor2 *)
        diHDry1Sensor3 : BOOL := 0;
        (* BOOL diHDry1Sensor3 *)
        diHDry1Sensor4 : BOOL := 0;
        (* BOOL diHDry1Sensor4 *)
        diHDry2Sensor1 : BOOL := 0;
        (* BOOL diHDry2Sensor1 *)
        diHDry2Sensor2 : BOOL := 0;
        (* BOOL diHDry2Sensor2 *)
        diHDry2Sensor3 : BOOL := 0;
        (* BOOL diHDry2Sensor3 *)
        diHDry2Sensor4 : BOOL := 0;
        (* BOOL diHDry2Sensor4 *)
        aiWaterLevel : REAL := 0.0;
        (* REAL aiWaterLevel *)

	END_STRUCT;

ComTCP_OUTPUTS_32BIT : STRUCT

		NumSignals	: INT := 53;

        doMaintenanceMode : BOOL := 0;
        (* BOOL doMaintenanceMode *)
        aoChemChemValve : REAL := 0.0;
        (* REAL aoChemChemValve *)
        doChemWaterValve : BOOL := 0;
        (* BOOL doChemWaterValve *)
        doChemRefill : BOOL := 0;
        (* BOOL doChemRefill *)
        doHighPressLiftRelay : BOOL := 0;
        (* BOOL doHighPressLiftRelay *)
        doHighPressLowerRelay : BOOL := 0;
        (* BOOL doHighPressLowerRelay *)
        doHighPressValve : BOOL := 0;
        (* BOOL doHighPressValve *)
        doHighPressPumpRelay : BOOL := 0;
        (* BOOL doHighPressPumpRelay *)
        doHBrushLiftRelay : BOOL := 0;
        (* BOOL doHBrushLiftRelay *)
        doHBrushLowerRelay : BOOL := 0;
        (* BOOL doHBrushLowerRelay *)
        doHBrushValve : BOOL := 0;
        (* BOOL doHBrushValve *)
        doHBrushBrushRelay : BOOL := 0;
        (* BOOL doHBrushBrushRelay *)
        doVBrushRelayLClose : BOOL := 0;
        (* BOOL doVBrushRelayLClose *)
        doVBrushRelayLOpen : BOOL := 0;
        (* BOOL doVBrushRelayLOpen *)
        doVBrushRelayRClose : BOOL := 0;
        (* BOOL doVBrushRelayRClose *)
        doVBrushRelayROpen : BOOL := 0;
        (* BOOL doVBrushRelayROpen *)
        aoVBrushLVel : REAL := 0.0;
        (* REAL aoVBrushLVel *)
        aoVBrushRVel : REAL := 0.0;
        (* REAL aoVBrushRVel *)
        doVBrushValve : BOOL := 0;
        (* BOOL doVBrushValve *)
        doVBrushRelayBrush : BOOL := 0;
        (* BOOL doVBrushRelayBrush *)
        doUnderbodyValve : BOOL := 0;
        (* BOOL doUnderbodyValve *)
        doUnderbodyPumpRelay : BOOL := 0;
        (* BOOL doUnderbodyPumpRelay *)
        doHPolishLiftRelay : BOOL := 0;
        (* BOOL doHPolishLiftRelay *)
        doHPolishLowerRelay : BOOL := 0;
        (* BOOL doHPolishLowerRelay *)
        doHPolishBrushRelay : BOOL := 0;
        (* BOOL doHPolishBrushRelay *)
        doVPolishRelayLClose : BOOL := 0;
        (* BOOL doVPolishRelayLClose *)
        doVPolishRelayLOpen : BOOL := 0;
        (* BOOL doVPolishRelayLOpen *)
        doVPolishRelayRClose : BOOL := 0;
        (* BOOL doVPolishRelayRClose *)
        doVPolishRelayROpen : BOOL := 0;
        (* BOOL doVPolishRelayROpen *)
        aoVPolishLVel : REAL := 0.0;
        (* REAL aoVPolishLVel *)
        aoVPolishRVel : REAL := 0.0;
        (* REAL aoVPolishRVel *)
        doVPolishRelayBrush : BOOL := 0;
        (* BOOL doVPolishRelayBrush *)
        doWaxValve : BOOL := 0;
        (* BOOL doWaxValve *)
        doWaxPumpRelay : BOOL := 0;
        (* BOOL doWaxPumpRelay *)
        doWaxRefill : BOOL := 0;
        (* BOOL doWaxRefill *)
        doHDry1LiftRelay : BOOL := 0;
        (* BOOL doHDry1LiftRelay *)
        doHDry1LowerRelay : BOOL := 0;
        (* BOOL doHDry1LowerRelay *)
        doHDry1VentRelay : BOOL := 0;
        (* BOOL doHDry1VentRelay *)
        doHDry1HeaterRelay : BOOL := 0;
        (* BOOL doHDry1HeaterRelay *)
        doVDry1VentRelay : BOOL := 0;
        (* BOOL doVDry1VentRelay *)
        doVDry1HeaterRelay : BOOL := 0;
        (* BOOL doVDry1HeaterRelay *)
        doHDry2LiftRelay : BOOL := 0;
        (* BOOL doHDry2LiftRelay *)
        doHDry2LowerRelay : BOOL := 0;
        (* BOOL doHDry2LowerRelay *)
        doHDry2VentRelay : BOOL := 0;
        (* BOOL doHDry2VentRelay *)
        doHDry2HeaterRelay : BOOL := 0;
        (* BOOL doHDry2HeaterRelay *)
        doConvRelay : BOOL := 0;
        (* BOOL doConvRelay *)
        doWaterValve : BOOL := 0;
        (* BOOL doWaterValve *)
        doTankWaterValve : BOOL := 0;
        (* BOOL doTankWaterValve *)
        doExitGreenLight : BOOL := 0;
        (* BOOL doExitGreenLight *)
        doExitOrangeLight : BOOL := 0;
        (* BOOL doExitOrangeLight *)
        doExitRedLight : BOOL := 0;
        (* BOOL doExitRedLight *)
        doExitLiftDoorRelay : BOOL := 0;
        (* BOOL doExitLiftDoorRelay *)
        doExitLowerDoorRelay : BOOL := 0;
        (* BOOL doExitLowerDoorRelay *)

	END_STRUCT;

END_TYPE
```

### MNG_Package.var
```iecst
(*                                                                            *)
(* File generated by the B&R AS 4 control config generator                    *)
(*                                                                            *)
(*     Provider: machineering                                                 *)
(*  Application: iPhysics_2.4.master                                          *)
(* Architecture: Windows 64 Bit                                               *)
(*      Version: 2.4.12706.master                                             *)
(*        Build: 608a88cb4                                                    *)
(*         Date: 2022-08-25, Time: 10:57:22                                   *)
(*                                                                            *)

                VAR
                ComTCP_SimInputs : ComTCP_INPUTS_32BIT := (0);
    ComTCP_SimOutputs : ComTCP_OUTPUTS_32BIT := (0);

    ComTCP_SimServerAddress : STRING[15] := '127.0.0.1';
    ComTCP_SimServerPort : UINT := 5000;
    ComTCP_SimSendCycleTime : TIME := T#20ms;
    ComTCP_SimActive : BOOL := FALSE;

                END_VAR
```

### MNG_Global.typ - Global data types
```iecst
TYPE
    (* 3d position *)
	VEC3 : STRUCT
		x: REAL;
		y: REAL;
		z: REAL;
	END_STRUCT;

	(* position and orientation as an euler based pose *)
	POSE6 :	STRUCT
		x: REAL;
		y: REAL;
		z: REAL;
		a: REAL;
		b: REAL;
		c: REAL;
	END_STRUCT;

	(* position and orientation as a 4x4 matrix *)
	TRAFO :STRUCT
		baseX : VEC3;
		fill0 : REAL;
		baseY : VEC3;
		fill1 : REAL;
		baseZ : VEC3;
		fill2 : REAL;
		origin : VEC3;
		fill3 : REAL;
	END_STRUCT;
END_TYPE
```

### Program Logical/Source/MainCtrl/MainCtrl (IEC)

#### Main.st - Init, cyclic, exit code
```iecst
PROGRAM _INIT

	//accessing structre and data from tasks
	Status1 	:= PV_xgetadr(ADR('EntryCtrl:iEntry'),ADR(EntryAddress),ADR(SizeEntry));
	Status2 	:= PV_xgetadr(ADR('ChemCtrl:iChem'),ADR(ChemAddress),ADR(SizeChem));
	Status3 	:= PV_xgetadr(ADR('Auxillary:iAuxillary'),ADR(AuxAddress),ADR(SizeAux));
	Status4		:= PV_xgetadr(ADR('HPWater:iHighPress'), ADR(HPAddress), ADR(SizeHP));
	Status5		:= PV_xgetadr(ADR('HBrushCtrl:iHBrush'), ADR(HBAddress), ADR(SizeHBrush));
	Status6		:= PV_xgetadr(ADR('HPolish:iHPolish'), ADR(HPolishAddress), ADR(SizeHPolish));
	Status7		:= PV_xgetadr(ADR('UBCtrl:iUBody'), ADR(UBodyAddress), ADR(SizeUBody));
	Status8		:= PV_xgetadr(ADR('WaxCtrl:iWax'), ADR(WaxAddress), ADR(SizeWax));
	Status9		:= PV_xgetadr(ADR('VBrushCtrl:iVBrush'), ADR(VBrushAddress), ADR(SizeVBrush));
	Status10	:= PV_xgetadr(ADR('VPolishCtr:iVPolish'), ADR(VPolishAddress), ADR(SizeVPolish));
	Status11	:= PV_xgetadr(ADR('DryHCtrl:iDry'), ADR(DryAddress), ADR(SizeDry));
	Status12	:= PV_xgetadr(ADR('DryH2Ctrl:iDry2'), ADR(Dry2Address), ADR(SizeDry2));

END_PROGRAM

PROGRAM _CYCLIC
	//accessing data from the addressZZ
	pEntryCtrl ACCESS EntryAddress;
	pChemCtrl ACCESS ChemAddress;
	pAuxCtrl ACCESS AuxAddress;
	pHPCtrl ACCESS HPAddress;
	pHBrushCtrl ACCESS HBAddress;
	pHPolish ACCESS HPolishAddress;
	pUBCtrl ACCESS UBodyAddress;
	pWaxCtrl ACCESS WaxAddress;
	pVBrush ACCESS VBrushAddress;
	pVPolish ACCESS VPolishAddress;
	pDry ACCESS DryAddress;
	pDry2 ACCESS Dry2Address;

	ScalDirt(x:=pEntryCtrl.IO.diSensSoilLvl ,y1:=5,x2:=10,y2:=0);

	IF gMain.Cmd.Start = TRUE THEN
		pAuxCtrl.doRelayConv	:= TRUE;
		gMain.Cmd.Start			:= FALSE;
		gMain.Option.EntryState	:= TRUE;
		iFl_CarFlag :=TRUE ;
	END_IF;

	IF (gMain.Option.EntryState = TRUE) THEN

		pEntryCtrl.Cmd.Start:=TRUE;
		txt:="entry";

		IF pEntryCtrl.IO.diSensEntry=TRUE THEN
			IF iFl_CarFlag =TRUE THEN
				FOR i:=0 TO 3 DO
					IF gCar[i]=FALSE THEN
						gCar[i]:=TRUE;
						iFb_Timer[i].IN:=TRUE;
						iFl_CarFlag :=FALSE;
						EXIT;
					END_IF;
				END_FOR;
			END_IF;
		END_IF;

	END_IF;

	IF iMi_Mode01 = TRUE THEN
		gMain.Option.EntryState		:= TRUE;
		gMain.Option.ChemicalState	:= TRUE;
		gMain.Option.HBrush			:= TRUE;
		gMain.Option.HighPress		:= TRUE;
		gMain.Option.Polish			:= TRUE;
		gMain.Option.UnderBody		:= TRUE;
		gMain.Option.VBrush			:= TRUE;
		gMain.Option.Wax			:= TRUE;
	END_IF;

	IF (iVa_Distance > 2.00) AND (gMain.Option.ChemicalState = TRUE) THEN	// chem station incoming
		gMain.Option.EntryState			:= FALSE;
		txt:="chem";
		pChemCtrl.IO.doChemWaterValve	:= TRUE;
	END_IF;

	IF (iVa_Distance > 7.5) THEN		// chem station outgoing (2.30 + 4.5)m
		pChemCtrl.IO.doChemWaterValve	:= FALSE;
		gMain.Option.ChemicalState		:= FALSE;
	END_IF;

	IF (iVa_Distance > 8.0) AND (gMain.Option.HighPress = TRUE) THEN
		txt:="HighPressure Water";
		pHPCtrl.Cmd.Start		:= TRUE;
	END_IF;

	IF (iVa_Distance > 13.50) AND (gMain.Option.HBrush = TRUE) THEN
		txt	:= "Horizontal Brush";
		pHBrushCtrl.Cmd.Start	:= TRUE;
		gMain.Option.HighPress	:= FALSE;
	END_IF;

	IF (iVa_Distance > 19.30) AND (gMain.Option.VBrush = TRUE) THEN
		txt	:= "Vertical Brush";
		pVBrush.Cmd.Start	:= TRUE;
		gMain.Option.HBrush		:= FALSE;
	END_IF;

	IF (iVa_Distance > 30.0) AND (gMain.Option.UnderBody = TRUE) THEN
		txt	:= "UnderBody Brush";
		pUBCtrl.Cmd.Start	:= TRUE;
		gMain.Option.VBrush	:= FALSE;
	END_IF;

	IF (iVa_Distance > 35.0) AND (gMain.Option.Polish = TRUE) THEN
		txt	:= "Polishing";
		pHPolish.Cmd.Start		:= TRUE;
		pVPolish.Cmd.Start		:= TRUE;
		gMain.Option.UnderBody	:= FALSE;
	END_IF;

	IF (iVa_Distance > 50.00) AND (gMain.Option.Wax = TRUE) THEN
		txt	:= "Waxing";
		pWaxCtrl.Cmd.Start	:= TRUE;
		gMain.Option.Polish	:= FALSE;
	END_IF;

	IF (iVa_Distance > 54.00) AND (gMain.Option.Dry = TRUE) THEN
		pDry.Cmd.Start		:= TRUE;
		pDry2.Cmd.Start		:= TRUE;
		gMain.Option.Wax	:= FALSE;
	END_IF;

	IF gMain.Cmd.EStop = TRUE THEN
		iFb_Timer[0]();
	END_IF;

END_PROGRAM

PROGRAM _EXIT
	(* Insert code here *)

END_PROGRAM
```

#### Types.typ - Local data types
```iecst
TYPE
	sMainStep_enum1 :
		( (*main enum*)
		enWAIT, (*wait state*)
		enSTART, (*start statre*)
		enENTRY, (*entry state*)
		enCHEMICAL (*chemical state*)
		);
END_TYPE
```

#### Variables.var - Local variables
```iecst
VAR
	ScalDirt : LCRScal;
	Status2 : UINT; (*status*)
	pEntryCtrl : REFERENCE TO EntryCtrl_typ; (*pointer*)
	SizeChem : UDINT; (*size of foil*)
	ChemAddress : UDINT; (*Address of foil*)
	pChemCtrl : REFERENCE TO ChemCtrl_typ; (*pointer*)
	txt : WSTRING[80]; (*text message*)
	SizeEntry : UDINT; (*size of foil*)
	EntryAddress : UDINT; (*Address of foil*)
	New_Variable : USINT; (*new variavle*)
	Car : INT; (*car is there *)
	Status3 : UINT; (*status*)
	Status1 : UINT; (*status*)
	i : INT; (*for loop*)
	SizeAux : UDINT; (*size of auxillary*)
	AuxAddress : UDINT; (*auxillary address*)
	pAuxCtrl : REFERENCE TO Auxillary_typ; (*auxillary pointer*)
	txt1 : WSTRING[80]; (*text*)
	iFb_Timer : ARRAY[0..2] OF TON := [3((PT:=T#147720ms))]; (*full timer*)
	Status4 : UINT; (*status*)
	HPAddress : UDINT; (*hp address*)
	SizeHP : UDINT; (*size of hp*)
	pHPCtrl : REFERENCE TO HPWaterCtrl_typ; (*hp pointer*)
	Status5 : UINT; (*status*)
	HBAddress : UDINT; (*hb address*)
	SizeHBrush : UDINT; (*size of brush*)
	pHBrushCtrl : REFERENCE TO HBrushCtrl_typ; (*pointer of hb*)
	Status6 : UINT; (*status*)
	HPolishAddress : UDINT; (*hp address*)
	SizeHPolish : UDINT; (*size of hp*)
	pHPolish : REFERENCE TO PolishCtrl_typ; (*hp pointer*)
	iFl_CarFlag : BOOL; (*flag if car is in or not*)
	Status7 : UINT; (*status *)
	UBodyAddress : UDINT; (*under body adr*)
	SizeUBody : UDINT; (*size of Ubody*)
	Status8 : UINT; (*status*)
	WaxAddress : UDINT; (*wax adr*)
	SizeWax : UDINT; (*size wax*)
	pUBCtrl : REFERENCE TO UBCtrl_typ; (*underbody control*)
	pWaxCtrl : REFERENCE TO WaxCtrl_typ; (*wax control*)
	Status9 : UINT; (*status*)
	VBrushAddress : UDINT; (*address of vb*)
	SizeVBrush : UDINT; (*size of vb*)
	pVBrush : REFERENCE TO VBrushCtrl_typ; (*vb pointer*)
	iVa_WaterLevel : REAL; (*water level*)
	iVa_WRefill : BOOL; (*water refill*)
	iVa_ChemLevel : REAL; (*chemical level*)
	iVa_ChemRefill : BOOL; (*chem refill*)
	iMi_Mode01 : BOOL; (*mode 1*)
	Status10 : UINT; (*statys*)
	VPolishAddress : UDINT; (*vp address*)
	SizeVPolish : UDINT; (*vp polish*)
	Status11 : UINT; (*status*)
	DryAddress : UDINT; (*dry address*)
	SizeDry : UDINT; (*size of dry*)
	pVPolish : REFERENCE TO VPolishCtrl_typ; (*pv polish*)
	pDry : REFERENCE TO DryCtrl_typ; (*pointer dry*)
	Status12 : UINT; (*status*)
	Dry2Address : UDINT; (*dry address*)
	SizeDry2 : UDINT; (*size of dry*)
	pDry2 : REFERENCE TO DryCtrl_typ; (*pointer dry*)
END_VAR
```

#### MainAlarm.st
```iecst
ACTION MainAlarm:

	IF iVa_WaterLevel<0.1 THEN
		MpAlarmXSet(gAlarmXCore,'WaterLow');
		IF MpAlarmXCheckReaction(gAlarmXCore, 'EStopErr') THEN
			gMain.Cmd.EStop:=TRUE;
		END_IF
	ELSE
		MpAlarmXReset(gAlarmXCore,'WaterLow');
	END_IF;

END_ACTION
```

### Program Logical/Source/Entrance/EntryCtrl (IEC)

#### Main.st - Init, cyclic, exit code
```iecst
PROGRAM _INIT
	(* Insert code here *)

END_PROGRAM

PROGRAM _CYCLIC
	(* Insert code here *)
	EntryAlarm;
	IF iEntry.Status.Error=TRUE THEN
		iEntryState:=enERROR;
	END_IF;

	CASE iEntryState OF

		enWAIT:
			iEntry.Status.Running:=FALSE ;
			IF iEntry.Cmd.Start=TRUE THEN
				iEntryState:=enSTART;
			END_IF;

		enSTART:
			iEntry.Status.Running:=TRUE ;
			IF iEntry.IO.diSensEntry=TRUE THEN
				iEntryState:=enCARIN;
			END_IF;
		enCARIN:
			iEntry.Status.CarIN:=TRUE;

			IF iEntry.IO.diSensEntry=FALSE THEN
				iEntry.Status.CarIN:=FALSE;
				iEntryState:=enWAIT;
			END_IF;

		enERROR:
			iEntry.Status.Running:=FALSE ;
			iEntry.Status.CarIN:=FALSE;
			iEntry.Cmd.Start:=FALSE;

			IF iEntry.Cmd.ErrorReset = TRUE THEN
				iEntry.Cmd.EStop:=FALSE;
				iEntry.Status.Error:=FALSE;
				iEntry.Cmd.ErrorReset:=FALSE;
				iEntryState:=enWAIT;
			END_IF;

	END_CASE;
END_PROGRAM

PROGRAM _EXIT
	(* Insert code here *)

END_PROGRAM
```

#### Types.typ - Local data types
```iecst
TYPE
	sStep :
		(
		enWAIT,
		enSTART,
		enCARIN,
		enERROR
		);
END_TYPE
```

#### Variables.var - Local variables
```iecst
VAR
	iEntry : EntryCtrl_typ;
	iEntryState : sStep;
END_VAR
```

#### EntryAlarm.st
```iecst
ACTION EntryAlarm:
	IF iEntry.Cmd.EStop=TRUE THEN
		MpAlarmXSet(gAlarmXCore,'EStopEntry');
		IF MpAlarmXCheckReaction(gAlarmXCore, 'EStopErr') THEN
			iEntry.Status.Error:= TRUE ;
		END_IF
	ELSE
		MpAlarmXReset(gAlarmXCore,'EStopEntry');
	END_IF;
END_ACTION
```

### EntryCtrl.typ
```iecst
TYPE
	EntryCmd_typ : 	STRUCT  (*command*)
		Start : BOOL; (*start command*)
		EStop : BOOL; (*estop command entry*)
		Stop : BOOL; (*stop command entry*)
		ErrorReset : BOOL; (*errorrest command entry*)
	END_STRUCT;
	EntryCtrl_typ : 	STRUCT  (*control main entry*)
		Cmd : EntryCmd_typ; (*command*)
		IO : EntryIOs_typ; (*IOs*)
		Par : EntryParam_typ; (*parameters*)
		Status : EntryStatus_typ; (*status*)
	END_STRUCT;
	EntryIOs_typ : 	STRUCT  (*IOs*)
		diSensEntry : BOOL; (*entry sens*)
		diSensSoilLvl : REAL; (*soil level*)
	END_STRUCT;
	EntryParam_typ : 	STRUCT  (*parameters*)
		CarLength : REAL; (*car length*)
	END_STRUCT;
	EntryStatus_typ : 	STRUCT  (*status*)
		Running : BOOL; (*running main control*)
		Error : BOOL; (*errror occured*)
		CarGone : BOOL; (*car gone*)
		CarIN : BOOL; (*car is in *)
	END_STRUCT;
END_TYPE
```

### Program Logical/Source/Chemicals/ChemCtrl (IEC)

#### Main.st - Init, cyclic, exit code
```iecst
PROGRAM _INIT
	(* Insert code here *)

END_PROGRAM

PROGRAM _CYCLIC
	(* Insert code here *)
	iChem.Par.ChemLevel:=ScalDirt.y;

	//if error then error state
	IF iChem.Status.Error=TRUE THEN
		sChemState:=enERROR;
	END_IF;

	CASE sChemState OF

		enWAIT:
			iChem.Status.Running:=FALSE;
			IF iChem.Cmd.Start= TRUE THEN
				sChemState:=enSPRAYON;
				iChem.Status.Running:=TRUE;
			END_IF;

		enSPRAYON:
			iChem.IO.doChemWaterValve	:=TRUE;
			iChem.Status.SprayON		:=TRUE ;
			IF iChem.IO.doChemWaterValve=FALSE THEN
				sChemState				:=enWAIT;
			END_IF;

		enERROR:
			iChem.Status.Running:=FALSE;
			iChem.IO.doChemWaterValve	:=FALSE;
			iChem.Status.SprayON		:=FALSE ;

			IF iChem.Cmd.ErrorReset=TRUE THEN
				iChem.Cmd.ErrorReset	:=FALSE;
				iChem.Cmd.EStop			:=FALSE;
				iChem.Status.Error		:=FALSE;
				sChemState				:=enWAIT;
			END_IF;

	END_CASE;
END_PROGRAM

PROGRAM _EXIT
	(* Insert code here *)

END_PROGRAM
```

#### Types.typ - Local data types
```iecst
TYPE
	sStep_enum :
		(
		enWAIT,
		enSPRAYON,
		enERROR
		);
END_TYPE
```

#### Variables.var - Local variables
```iecst
VAR
	sChemState : sStep_enum;
	ScalDirt : LCRScal;
	iChem : ChemCtrl_typ;
END_VAR
```

#### ChemAlarm.st
```iecst
ACTION ChemAlarm:
	IF iChem.Cmd.EStop=TRUE THEN
		MpAlarmXSet(gAlarmXCore,'EStopChem');
		IF MpAlarmXCheckReaction(gAlarmXCore, 'EStopErr') THEN
			iChem.Status.Error:= TRUE ;
		END_IF
	ELSE
		MpAlarmXReset(gAlarmXCore,'EStopChem');
	END_IF;

	IF iChem.Par.ChemLevel	<0.1 THEN
		MpAlarmXSet(gAlarmXCore,'ChemLow');
		iChem.Status.Error	:=TRUE ;
	ELSE
		MpAlarmXReset(gAlarmXCore,'ChemLow');
		iChem.Cmd.ChemRefill:= FALSE ;
	END_IF;
	IF iChem.Cmd.ChemRefill	=TRUE THEN
		iChem.Status.Error	:=TRUE ;
		iChem.Cmd.ErrorReset:=TRUE;
		iChem.Cmd.ChemRefill:=FALSE;
	END_IF;

END_ACTION
```

### ChemCtrl.typ
```iecst
TYPE
	ChemCmd_typ : 	STRUCT
		Start : BOOL;
		EStop : BOOL;
		Stop : BOOL;
		ErrorReset : BOOL;
		ChemRefill : BOOL;
	END_STRUCT;
	ChemCtrl_typ : 	STRUCT
		Cmd : ChemCmd_typ;
		IO : ChemIOs_typ;
		Par : ChemParam_typ;
		Status : ChemStatus_typ;
	END_STRUCT;
	ChemIOs_typ : 	STRUCT
		aoChemChemValve : REAL;
		doChemWaterValve : BOOL;
		doChemRefill : BOOL;
	END_STRUCT;
	ChemParam_typ : 	STRUCT
		ChemLevel : REAL;
	END_STRUCT;
	ChemStatus_typ : 	STRUCT
		Running : BOOL;
		Error : BOOL;
		ChemHigh : BOOL;
		ChemLow : BOOL;
		SprayON : BOOL;
	END_STRUCT;
END_TYPE
```

### Program Logical/Source/HPWater/HPWater (IEC)

#### Types.typ
```iecst
TYPE
	HighPressureState_enum :
		(
		enWAIT,
		enSTART,
		enOPERATION,
		enERROR
		);
END_TYPE
```

#### Variables.var
```iecst
VAR
	sHighPressState : HighPressureState_enum; (*enumeration*)
	iHighPress : HPWaterCtrl_typ; (*main control*)
END_VAR
```

#### HPAlarm.st
```iecst
ACTION EStopHighPre:
	IF iHighPress.Cmd.EStop=TRUE THEN
		MpAlarmXSet(gAlarmXCore,'EStopHighPre');
		IF MpAlarmXCheckReaction(gAlarmXCore, 'EStopErr') THEN
			iHighPress.Status.Error:= TRUE ;
		END_IF
	ELSE
		MpAlarmXReset(gAlarmXCore,'EStopHighPre');
	END_IF;
END_ACTION
```

#### Main.st
```iecst
PROGRAM _INIT
	(* Insert code here *)

END_PROGRAM

PROGRAM _CYCLIC
	(* Insert code here *)
	EStopHighPre;
	CASE sHighPressState OF
		enWAIT:
			IF iHighPress.Cmd.Start = TRUE THEN
				sHighPressState				:= enSTART;
				iHighPress.IO.doValveHP		:= TRUE;
			END_IF;
		enSTART:
			IF (iHighPress.IO.diSensHP1 = FALSE) AND (iHighPress.IO.diSensHP2 = FALSE) AND (iHighPress.IO.diSensHP3 = FALSE) AND (iHighPress.IO.diSensHP4 = FALSE) THEN
				iHighPress.IO.doRelayHPLow	:= TRUE;
				iHighPress.IO.doRelayHPLift	:= FALSE;
			END_IF;
			IF (iHighPress.IO.diSensHP1 = TRUE) AND (iHighPress.IO.diSensHP2 = FALSE) AND (iHighPress.IO.diSensHP3 = FALSE) AND (iHighPress.IO.diSensHP4 = FALSE) THEN
				iHighPress.IO.doRelayHPLow	:= FALSE;
				iHighPress.IO.doRelayHPLift	:= FALSE;
				iHighPress.IO.doRelayHPPump	:= TRUE;
				sHighPressState				:= enOPERATION;
			END_IF;

		enOPERATION:
			IF (iHighPress.IO.diSensHP1 = TRUE) AND (iHighPress.IO.diSensHP2 = FALSE) AND (iHighPress.IO.diSensHP3 = FALSE) AND (iHighPress.IO.diSensHP4 = FALSE) THEN
				iHighPress.IO.doRelayHPLow	:= FALSE;
				iHighPress.IO.doRelayHPLift	:= FALSE;
			END_IF;
			IF (iHighPress.IO.diSensHP1 = TRUE) AND (iHighPress.IO.diSensHP2 = TRUE) AND (iHighPress.IO.diSensHP3 = TRUE) AND (iHighPress.IO.diSensHP4 = FALSE) THEN
				iHighPress.IO.doRelayHPLow	:= FALSE;
				iHighPress.IO.doRelayHPLift	:= TRUE;
			END_IF;
			IF (iHighPress.IO.diSensHP1 = TRUE) AND (iHighPress.IO.diSensHP2 = TRUE) AND (iHighPress.IO.diSensHP3 = FALSE) AND (iHighPress.IO.diSensHP4 = FALSE) THEN
				iHighPress.IO.doRelayHPLow	:= FALSE;
				iHighPress.IO.doRelayHPLift	:= TRUE;
			END_IF;
			IF (iHighPress.IO.diSensHP1 = FALSE) AND (iHighPress.IO.diSensHP2 = FALSE) AND (iHighPress.IO.diSensHP3 = TRUE) AND (iHighPress.IO.diSensHP4 = FALSE) THEN
				iHighPress.IO.doRelayHPLow	:= TRUE;
				iHighPress.IO.doRelayHPLift	:= FALSE;
			END_IF;
			IF (iHighPress.IO.diSensHP1 = FALSE) AND (iHighPress.IO.diSensHP2 = FALSE) AND (iHighPress.IO.diSensHP3 = TRUE) AND (iHighPress.IO.diSensHP4 = TRUE) THEN
				iHighPress.IO.doRelayHPLow	:= FALSE;
				iHighPress.IO.doRelayHPLift	:= FALSE;
			END_IF;
			IF (iHighPress.IO.diSensHP1 = FALSE) AND (iHighPress.IO.diSensHP2 = FALSE) AND (iHighPress.IO.diSensHP3 = FALSE) AND (iHighPress.IO.diSensHP4 = FALSE) THEN
				iHighPress.IO.doRelayHPLow	:= FALSE;
				iHighPress.IO.doRelayHPLift	:= FALSE;
				iHighPress.IO.doRelayHPPump	:= FALSE;
				iHighPress.IO.doValveHP		:= FALSE;
				iHighPress.Cmd.Start		:= FALSE;
				sHighPressState				:= enWAIT;
			END_IF;

		enERROR:
			iHighPress.IO.doRelayHPLow	:= FALSE;
			iHighPress.IO.doRelayHPLift	:= FALSE;
			iHighPress.IO.doRelayHPPump	:= FALSE;
			iHighPress.IO.doValveHP		:= FALSE;
			iHighPress.Cmd.Start		:= FALSE;

			IF iHighPress.Cmd.ErrorReset = TRUE THEN
				iHighPress.Cmd.EStop:=FALSE;
				iHighPress.Status.Error:=FALSE;
				iHighPress.Cmd.ErrorReset:=FALSE;
				sHighPressState:=enWAIT;
			END_IF;

	END_CASE;

END_PROGRAM

PROGRAM _EXIT
	(* Insert code here *)

END_PROGRAM
```

### HPWater.typ
```iecst
TYPE
	HPWaterCmd_typ : 	STRUCT  (*water command*)
		Start : BOOL; (*command start*)
		EStop : BOOL; (*estop command*)
		Stop : BOOL; (*stop command*)
		ErrorReset : USINT; (*command error reset*)
	END_STRUCT;
	HPWaterCtrl_typ : 	STRUCT  (*main ocntrol OF HPWater*)
		Cmd : HPWaterCmd_typ; (*command OF HPWater*)
		IO : HPWaterIOs_typ; (*ios OF HPWater*)
		Par : HPWaterParam_typ; (*parameters*)
		Status : HPWaterStatus_typ; (*stauts OF HPWater*)
	END_STRUCT;
	HPWaterIOs_typ : 	STRUCT  (*water ios*)
		diSensHP1 : BOOL; (*sesnsor 1 OF HPWater*)
		diSensHP2 : BOOL; (*sensor 2 OF HPWater*)
		diSensHP3 : BOOL; (*sensor 3 OF HPWater*)
		diSensHP4 : BOOL; (*sensor 4 OF HPWater*)
		doValveHP : BOOL; (*valve of hp*)
		doRelayHPPump : BOOL; (*relay fro pump*)
		doRelayHPLow : BOOL; (*lowering bar*)
		doRelayHPLift : BOOL; (*lifting bar*)
	END_STRUCT;
	HPWaterParam_typ : 	STRUCT  (*parameters OF HPWater*)
		New_Member : USINT;
	END_STRUCT;
	HPWaterStatus_typ : 	STRUCT  (*water status OF HPWater*)
		Running : BOOL; (*running OF HPWater*)
		Error : BOOL; (*error OF HPWater*)
		ValveOpen : USINT; (*valve open OF HPWater*)
	END_STRUCT;
END_TYPE
```

### Program Logical/Source/HBrush/HBrushCtrl (IEC)

#### Main.st - Init, cyclic, exit code
```iecst
PROGRAM _INIT
	(* Insert code here *)

END_PROGRAM

PROGRAM _CYCLIC
	(* Insert code here *)
	EStopHB;
	CASE sHBrushState OF
		enWAIT:
			IF iHBrush.Cmd.Start = TRUE THEN
				sHBrushState				:= enSTART;
			END_IF;
		enSTART:
			IF (iHBrush.IO.diSensHB1 = FALSE) AND (iHBrush.IO.diSensHB2 = FALSE) AND (iHBrush.IO.diSensHB3 = FALSE) AND (iHBrush.IO.diSensHB4 = FALSE) THEN
				iHBrush.IO.doRelayHBLower	:= TRUE;
				iHBrush.IO.doRelayHBLift	:= FALSE;
			END_IF;
			IF (iHBrush.IO.diSensHB1 = TRUE) AND (iHBrush.IO.diSensHB2 = FALSE) AND (iHBrush.IO.diSensHB3 = FALSE) AND (iHBrush.IO.diSensHB4 = FALSE) THEN
				iHBrush.IO.doRelayHBLower	:= FALSE;
				iHBrush.IO.doRelayHBLift	:= FALSE;
				iHBrush.IO.doRelayHBBrush	:= TRUE;
				iHBrush.IO.doValveHB		:= TRUE;
				sHBrushState				:= enOPERATION;
			END_IF;
		enOPERATION:
			IF (iHBrush.IO.diSensHB1 = TRUE) AND (iHBrush.IO.diSensHB2 = FALSE) AND (iHBrush.IO.diSensHB3 = FALSE) AND (iHBrush.IO.diSensHB4 = FALSE) THEN
				iHBrush.IO.doRelayHBLower	:= FALSE;
				iHBrush.IO.doRelayHBLift	:= FALSE;
			END_IF;
			IF (iHBrush.IO.diSensHB1 = TRUE) AND (iHBrush.IO.diSensHB2 = TRUE) AND (iHBrush.IO.diSensHB3 = TRUE) AND (iHBrush.IO.diSensHB4 = FALSE) THEN
				iHBrush.IO.doRelayHBLower	:= FALSE;
				iHBrush.IO.doRelayHBLift	:= TRUE;
			END_IF;
			IF (iHBrush.IO.diSensHB1 = TRUE) AND (iHBrush.IO.diSensHB2 = TRUE) AND (iHBrush.IO.diSensHB3 = FALSE) AND (iHBrush.IO.diSensHB4 = FALSE) THEN
				iHBrush.IO.doRelayHBLower	:= FALSE;
				iHBrush.IO.doRelayHBLift	:= TRUE;
			END_IF;
			IF (iHBrush.IO.diSensHB1 = FALSE) AND (iHBrush.IO.diSensHB2 = FALSE) AND (iHBrush.IO.diSensHB3 = TRUE) AND (iHBrush.IO.diSensHB4 = FALSE) THEN
				iHBrush.IO.doRelayHBLower	:= TRUE;
				iHBrush.IO.doRelayHBLift	:= FALSE;
			END_IF;
			IF (iHBrush.IO.diSensHB1 = FALSE) AND (iHBrush.IO.diSensHB2 = FALSE) AND (iHBrush.IO.diSensHB3 = TRUE) AND (iHBrush.IO.diSensHB4 = TRUE) THEN
				iHBrush.IO.doRelayHBLower	:= FALSE;
				iHBrush.IO.doRelayHBLift	:= FALSE;
			END_IF;
			IF (iHBrush.IO.diSensHB1 = FALSE) AND (iHBrush.IO.diSensHB2 = FALSE) AND (iHBrush.IO.diSensHB3 = FALSE) AND (iHBrush.IO.diSensHB4 = FALSE) THEN
				iHBrush.IO.doRelayHBLower	:= FALSE;
				iHBrush.IO.doRelayHBLift	:= FALSE;
				iHBrush.IO.doRelayHBBrush	:= FALSE;
				iHBrush.IO.doValveHB		:= FALSE;
				iHBrush.Cmd.Start			:= FALSE;
				sHBrushState				:= enWAIT;
			END_IF;

		enERROR:
			iHBrush.IO.doRelayHBLower	:= FALSE;
			iHBrush.IO.doRelayHBLift	:= FALSE;
			iHBrush.IO.doRelayHBBrush	:= FALSE;
			iHBrush.IO.doValveHB		:= FALSE;
			iHBrush.Cmd.Start			:= FALSE;

			IF iHBrush.Cmd.ErrorReset = TRUE THEN
				iHBrush.Cmd.EStop:=FALSE;
				iHBrush.Status.Error:=FALSE;
				iHBrush.Cmd.ErrorReset:=FALSE;
				sHBrushState:=enWAIT;
			END_IF;
	END_CASE;

END_PROGRAM

PROGRAM _EXIT
	(* Insert code here *)

END_PROGRAM
```

#### Types.typ - Local data types
```iecst
TYPE
	HorizonBrushState_enum :
		(
		enWAIT,
		enSTART,
		enOPERATION,
		enERROR
		);
END_TYPE
```

#### Variables.var - Local variables
```iecst
VAR
	iHBrush : HBrushCtrl_typ; (*hb brush*)
	sHBrushState : HorizonBrushState_enum; (*enumeration*)
	iDry : DryCtrl_typ; (*local dry main str*)
END_VAR
```

#### HBAlarm.st
```iecst
ACTION EStopHB:
	IF iHBrush.Cmd.EStop=TRUE THEN
		MpAlarmXSet(gAlarmXCore,'EStopHB');
		IF MpAlarmXCheckReaction(gAlarmXCore, 'EStopErr') THEN
			iHBrush.Status.Error:= TRUE ;
		END_IF
	ELSE
		MpAlarmXReset(gAlarmXCore,'EStopHB');
	END_IF;
END_ACTION
```

### HBrushCtrl.typ
```iecst
TYPE
	HBrushCmd_typ : 	STRUCT  (*hb command*)
		Start : BOOL; (*start command*)
		EStop : BOOL; (*estop command*)
		Stop : BOOL; (*stop command*)
		ErrorReset : USINT; (*error reset command*)
	END_STRUCT;
	HBrushCtrl_typ : 	STRUCT  (*control  of HBRUSH*)
		Cmd : HBrushCmd_typ; (*command of HBRUSH*)
		IO : HBrushIOs_typ; (*IOs of HBRUSH*)
		Par : HBrushParam_typ; (*parameters of HBRUSH*)
		Status : HBrushStatus_typ; (*statsus of HBRUSH*)
	END_STRUCT;
	HBrushIOs_typ : 	STRUCT  (*IOs of HBRUSH*)
		doRelayHBLift : BOOL; (*lifting HB of HBRUSH*)
		doRelayHBLower : BOOL; (*lowring HB of HBRUSH*)
		doRelayHBBrush : BOOL; (*Brush relay of HBRUSH*)
		doValveHB : BOOL; (*valve relay of HBRUSH*)
		diSensHB2 : BOOL; (*sensor1 of HBRUSH*)
		diSensHB3 : BOOL; (*sensor 2 of HBRUSH*)
		diSensHB4 : BOOL; (*sensor 3 of HBRUSH*)
		diSensHB1 : BOOL; (*sensor 4 of HBRUSH*)
	END_STRUCT;
	HBrushParam_typ : 	STRUCT  (*parameters of HBRUSH*)
		VehHeight : REAL; (*height of vehicle*)
	END_STRUCT;
	HBrushStatus_typ : 	STRUCT  (*status of HBRUSH*)
		Running : BOOL; (*running  of HBRUSH*)
		Error : BOOL; (*error of HBRUSH*)
		Lifting : BOOL; (*lifting of HBRUSH*)
		Brushing : BOOL; (*brushing  of HBRUSH*)
		ValveOpen : BOOL; (*valve open  of HBRUSH*)
		Lowering : BOOL; (*lowering  of HBRUSH*)
	END_STRUCT;
END_TYPE
```

### Program Logical/Source/VBrush/VBrushCtrl (IEC)

#### Main.st - Init, cyclic, exit code
```iecst
PROGRAM _INIT
	(* Insert code here *)

END_PROGRAM

PROGRAM _CYCLIC
	(* Insert code here *)
	VBAlarm;
	IF iVBrush.Status.Error=TRUE THEN
		sVBrushState:=enERROR;
	END_IF;

	CASE sVBrushState OF

		enWAIT:

			IF iVBrush.Cmd.Start=TRUE THEN
				sVBrushState:=enSTART;
			END_IF;

		enSTART:
			iVBrush.IO.doRelayVBLClose:=TRUE;
			iVBrush.IO.doRelayVBRClose:=TRUE;
			IF (iVBrush.IO.aiVBLForceF > 70.0) AND (iVBrush.IO.aiVBRForceF  > 70.0) THEN
				iVBrush.IO.doRelayVBLClose	:=FALSE;
				iVBrush.IO.doRelayVBRClose	:=FALSE;
				sVBrushState:=enOPEN;
			END_IF;

		enOPEN:
			iVBrush.IO.doRelayVBROpen :=TRUE;
			iVBrush.IO.doRelayVBLOpen :=TRUE;
			IF (iVBrush.IO.aiVBLForceF <= 5.0) AND (iVBrush.IO.aiVBRForceF <= 5.0 ) THEN
				iVBrush.IO.doRelayVBROpen :=FALSE;
				iVBrush.IO.doRelayVBLOpen :=FALSE;
				sVBrushState:=enCLOSE;
			END_IF;

		enCLOSE:
			iVBrush.IO.doRelayVBLClose:=TRUE;
			iVBrush.IO.doRelayVBRClose:=TRUE;

			IF (iVBrush.IO.aiVBLForceS > 120) AND (iVBrush.IO.aiVBRForceS > 120) THEN
				sVBrushState:=enOPERATION;
			END_IF;

		enOPERATION:
			iVBrush.IO.doRelayVBLClose:=FALSE;
			iVBrush.IO.doRelayVBRClose:=FALSE;
			IF (iVBrush.IO.aiVBLForceS =0 AND iVBrush.IO.aiVBRForceS =0) THEN
				sVBrushState:=enSTART;
			END_IF;

		enERROR:
			iVBrush.IO.doRelayVBLClose:=FALSE;
			iVBrush.IO.doRelayVBRClose:=FALSE;
			iVBrush.IO.doRelayVBROpen :=FALSE;
			iVBrush.IO.doRelayVBLOpen :=FALSE;
			IF iVBrush.Cmd.ErrorReset=TRUE THEN
				iVBrush.Cmd.ErrorReset:=FALSE;
				iVBrush.Status.Error:=FALSE;
				sVBrushState:=enSTART;
			END_IF;

	END_CASE;
END_PROGRAM

PROGRAM _EXIT
	(* Insert code here *)

END_PROGRAM
```

#### Variables.var - Local variables
```iecst
VAR
	iVBrush : VBrushCtrl_typ; (*brush main control*)
	sVBrushState : sStep_enum; (*vb enumeration*)
END_VAR
```

#### VBAlarm.st
```iecst
ACTION VBAlarm:
	IF iVBrush.Cmd.EStop=TRUE THEN
		MpAlarmXSet(gAlarmXCore,'EStopVB');
		IF MpAlarmXCheckReaction(gAlarmXCore, 'EStopErr') THEN
			iVBrush.Status.Error:= TRUE ;
		END_IF
	ELSE
		MpAlarmXReset(gAlarmXCore,'EStopVB');
	END_IF;
END_ACTION
```

### VBrushCtrl.typ
```iecst
TYPE
	VBrushCmd_typ : 	STRUCT  (*commands*)
		Start : BOOL; (*start of Vbrush*)
		EStop : BOOL; (*estop of Vbrush*)
		Stop : BOOL; (*stop  of Vbrush*)
		ErrorReset : USINT; (* error reseet of Vbrush*)
	END_STRUCT;
	VBrushCtrl_typ : 	STRUCT  (*control*)
		Cmd : VBrushCmd_typ; (*commands*)
		IO : VBrushIOs_typ; (*ios  of Vbrush*)
		Par : VBrushParam_typ; (*parameteres  of Vbrush*)
		Status : VBrushStatus_typ; (*status  of Vbrush*)
	END_STRUCT;
	VBrushIOs_typ : 	STRUCT  (*ios*)
		doRelayVBLClose : BOOL; (*leftcloseof Vbrush*)
		doRelayVBROpen : BOOL; (*rightopen of Vbrush*)
		doRelayVBLOpen : BOOL; (*leftopen of Vbrush*)
		doRelayVBRClose : BOOL; (*rightclose of Vbrush*)
		aiVBRForceS : REAL; (*sideforce of Vbrush*)
		aiVBRForceF : REAL; (*frontforce of Vbrush*)
		aiVBLForceS : REAL; (*sideforce of Vbrush*)
		aiVBLForceF : REAL; (*leftforce of Vbrush*)
		aoVBRRVelocity : REAL; (*velocity*)
		aoVBRLVelocity : REAL; (*velocity*)
	END_STRUCT;
	VBrushParam_typ : 	STRUCT
		LeftVel : REAL := 5.0; (*leftvelocity*)
		RightVel : REAL := 5.0; (*rightvelocity*)
	END_STRUCT;
	VBrushStatus_typ : 	STRUCT
		Running : BOOL; (*running of Vbrush*)
		Error : BOOL; (*error  of Vbrush*)
		ForceIN : BOOL; (*forcein of Vbrush*)
		Rotating : USINT; (*rotating of Vbrush*)
	END_STRUCT;
END_TYPE
```

### Program Logical/Source/OptUnderBody/UBCtrl (IEC)

#### Main.st - Init, cyclic, exit code
```iecst
PROGRAM _INIT
	(* Insert code here *)

END_PROGRAM

PROGRAM _CYCLIC
	(* Insert code here *)

	UBAlarm;
	IF iUBody.Status.Error=TRUE THEN
		iUBodyState:=enERROR;
	END_IF;

	CASE iUBodyState OF

		enWAIT:
			iUBody.IO.doRelayPump:=FALSE;
			iUBody.IO.doValveUB:=FALSE;
			iUBody.Status.ValveOpen:=FALSE;
			iUBody.Status.PumpOpen:=FALSE;
			IF iUBody.Cmd.Start=TRUE THEN
				iUBodyState:=enUBODYON;
			END_IF;

		enUBODYON:
			iUBody.IO.doRelayPump:=TRUE;
			iUBody.IO.doValveUB:=TRUE;
			iUBody.Status.ValveOpen:=TRUE;
			iUBody.Status.PumpOpen:=TRUE;

			IF iUBody.IO.doValveUB = FALSE THEN
				iUBodyState:=enWAIT;
			END_IF;
		enERROR:
			iUBody.IO.doRelayPump		:=FALSE;
			iUBody.IO.doValveUB			:=FALSE;
			iUBody.Status.ValveOpen		:=FALSE;
			iUBody.Status.PumpOpen		:=FALSE;
			IF iUBody.Cmd.ErrorReset 	= TRUE THEN
				iUBody.Cmd.ErrorReset 	:= FALSE;
				iUBody.Status.Error		:=FALSE;
				iUBody.Cmd.EStop		:=FALSE;
				iUBodyState				:=enWAIT;
			END_IF;
	END_CASE;
END_PROGRAM

PROGRAM _EXIT
	(* Insert code here *)

END_PROGRAM
```

#### Types.typ - Local data types
```iecst
TYPE
	sStep :
		(
		enWAIT,
		enUBODYON,
		enERROR
		);
END_TYPE
```

#### Variables.var - Local variables
```iecst
VAR
	iUBody : UBCtrl_typ; (*underbody main control*)
	iUBodyState : sStep; (*enum main*)
END_VAR
```

#### UBAlarm.st
```iecst
ACTION UBAlarm:
	IF iUBody.Cmd.EStop=TRUE THEN
		MpAlarmXSet(gAlarmXCore,'EStopUB');
		IF MpAlarmXCheckReaction(gAlarmXCore, 'EStopErr') THEN
			iUBody.Status.Error:= TRUE ;
		END_IF
	ELSE
		MpAlarmXReset(gAlarmXCore,'EStopUB');
	END_IF;
END_ACTION
```

### UBCtrl.typ
```iecst
TYPE
	UBCmd_typ : 	STRUCT  (*commmand of UBody*)
		Start : BOOL; (*start of UBody*)
		EStop : BOOL; (*estop of UBody*)
		Stop : BOOL; (*stop of UBody*)
		ErrorReset : USINT; (*errorrest of UBody*)
	END_STRUCT;
	UBCtrl_typ : 	STRUCT  (*control  of UBody*)
		Cmd : UBCmd_typ; (*command of UBody*)
		IO : UBIOs_typ; (*IOs  of UBody*)
		Par : UBParam_typ; (*parameters*)
		Status : UBStatus_typ; (*parametes of UBody*)
	END_STRUCT;
	UBIOs_typ : 	STRUCT  (*IOs*)
		doValveUB : BOOL; (*valve is on*)
		doRelayPump : BOOL; (*relay is on*)
	END_STRUCT;
	UBParam_typ : 	STRUCT
		New_Member : USINT;
	END_STRUCT;
	UBStatus_typ : 	STRUCT  (*status*)
		Running : BOOL; (*running  of UBody*)
		Error : BOOL; (*error of UBody*)
		PumpOpen : BOOL; (*pump of UBody*)
		ValveOpen : BOOL; (*valve of UBody*)
	END_STRUCT;
END_TYPE
```

### Program Logical/Source/OptVpolish/VPolishCtr (IEC)

#### Main.st - Init, cyclic, exit code
```iecst
PROGRAM _INIT
	(* Insert code here *)
	iVPolish.IO.aoVPLVel:=5;
	iVPolish.IO.aoVPRVel:=5;

END_PROGRAM

PROGRAM _CYCLIC
	(* Insert code here *)
	VPolAlarm;
	IF iVPolish.Status.Error=TRUE THEN
		sVPolishState :=enERROR;
	END_IF;

	CASE sVPolishState OF

		enWAIT:

			IF iVPolish.Cmd.Start=TRUE THEN
				sVPolishState:=enSTART;
			END_IF;

		enSTART:
			iVPolish.IO.doRelayRClose 		:=TRUE;
			iVPolish.IO.doRelayLClose		:=TRUE;
			IF (iVPolish.IO.aiVPLForceF > 70.0) AND (iVPolish.IO.aiVPRForceF  > 70.0) THEN
				iVPolish.IO.doRelayRClose	:=FALSE;
				iVPolish.IO.doRelayLClose	:=FALSE;
				sVPolishState:=enOPEN;
			END_IF;

		enOPEN:
			iVPolish.IO.doRelayLOpen :=TRUE;
			iVPolish.IO.doRelayROpen :=TRUE;
			IF (iVPolish.IO.aiVPLForceF <= 5.0) AND (iVPolish.IO.aiVPRForceF <= 5.0 ) THEN
				iVPolish.IO.doRelayLClose :=FALSE;
				iVPolish.IO.doRelayRClose :=FALSE;
				sVPolishState:=enCLOSE;
			END_IF;
			//	(iVPolish.IO.aiVBLForceS >120 AND iVPolish.IO.aiVBRForceS >120)

		enCLOSE:
			iVPolish.IO.doRelayRClose:=TRUE;
			iVPolish.IO.doRelayLClose:=TRUE;

			IF (iVPolish.IO.aiVPLForceS > 120) AND (iVPolish.IO.aiVPRForceS > 120) THEN
				sVPolishState:=enOPERATION;
			END_IF;

		enOPERATION:
			iVPolish.IO.doRelayRClose:=FALSE;
			iVPolish.IO.doRelayLClose:=FALSE;
			IF (iVPolish.IO.aiVPLForceS =0 AND iVPolish.IO.aiVPRForceS =0) THEN
				sVPolishState:=enSTART;
			END_IF;

		enERROR:
			iVPolish.IO.doRelayLClose:=FALSE;
			iVPolish.IO.doRelayRClose:=FALSE;
			iVPolish.IO.doRelayRClose:=FALSE;
			iVPolish.IO.doRelayLClose:=FALSE;

			IF iVPolish.Cmd.ErrorReset=TRUE THEN
				iVPolish.Status.Error:=FALSE;
				iVPolish.Cmd.EStop	 :=FALSE;
				iVPolish.Cmd.ErrorReset:=FALSE;
				sVPolishState:=enSTART;
			END_IF;

	END_CASE;
END_PROGRAM

PROGRAM _EXIT
	(* Insert code here *)

END_PROGRAM
```

#### Types.typ - Local data types
```iecst
TYPE
	sStep_enum :
		(
		enWAIT,
		enSTART,
		enOPEN,
		enCLOSE,
		enOPERATION,
		enERROR
		);
END_TYPE
```

#### Variables.var - Local variables
```iecst
VAR
	iVPolish : VPolishCtrl_typ; (*main vp control*)
	sVPolishState : sStep_enum; (*enum of polsih*)
END_VAR
```

#### VPAlarm.st
```iecst
ACTION VPolAlarm:
	IF iVPolish.Cmd.EStop=TRUE THEN
		MpAlarmXSet(gAlarmXCore,'EStopVPol');
		IF MpAlarmXCheckReaction(gAlarmXCore, 'EStopErr') THEN
			iVPolish.Status.Error:= TRUE ;
		END_IF
	ELSE
		MpAlarmXReset(gAlarmXCore,'EStopVPol');
	END_IF;
END_ACTION
```

### VPolishCtrl.typ
```iecst
TYPE
	VPolishCmd_typ : 	STRUCT  (*commanding*)
		Start : BOOL; (*start vpolish*)
		EStop : BOOL; (*estop  of UBody*)
		Stop : BOOL; (*stop of vpolish*)
		ErrorReset : USINT; (* error reset of vpolish*)
	END_STRUCT;
	VPolishCtrl_typ : 	STRUCT  (*control*)
		Cmd : VPolishCmd_typ; (*command  of vpolish*)
		IO : VPolishIOs_typ; (*IO  of vpolish*)
		Status : VPolishStatus_typ; (*status of vpolish*)
	END_STRUCT;
	VPolishIOs_typ : 	STRUCT  (*IOs  of vpolish*)
		doRelayRClose : BOOL; (*realy close  of vpolish*)
		doRelayROpen : BOOL; (*relay  of vpolish*)
		doRelayLClose : BOOL; (*relay  of vpolish*)
		doRelayLOpen : BOOL; (*left oepn  of vpolish*)
		doRelayBrush : BOOL; (*relay brush  of vpolish*)
		aoVPLVel : REAL; (*right valve  of vpolish*)
		aoVPRVel : REAL; (*Right vel  of vpolish*)
		aiVPRForceS : REAL; (*sideforce of vpolish*)
		aiVPRForceF : REAL; (*force front  of vpolish*)
		aiVPLForceS : REAL; (*side of vpolish*)
		aiVPLForceF : REAL; (*force front  of vpolish*)
	END_STRUCT;
	VPolishStatus_typ : 	STRUCT  (*status*)
		Running : BOOL; (*running  of vpolish*)
		Error : BOOL; (*error of vpolish*)
		ForceIN : USINT; (*forcein of vpolish*)
		Rotating : USINT; (*rotating of vpolish*)
	END_STRUCT;
END_TYPE
```

### Program Logical/Source/OptVpolish/VPolishCtrl

#### Main.st
```iecst
PROGRAM _INIT
	(* Insert code here *)

END_PROGRAM

PROGRAM _CYCLIC
	(* Insert code here *)
	VPolAlarm;
	IF iVPolish.Status.Error=TRUE THEN
		sVPolishState :=enERROR;
	END_IF;

	CASE sVPolishState OF

		enWAIT:

			IF iVPolish.Cmd.Start=TRUE THEN
				sVPolishState:=enSTART;
			END_IF;

		enSTART:
			iVPolish.IO.doRelayRClose 		:=TRUE;
			iVPolish.IO.doRelayLClose		:=TRUE;
			IF (iVPolish.IO.aiVPLForceF > 70.0) AND (iVPolish.IO.aiVPRForceF  > 70.0) THEN
				iVPolish.IO.doRelayRClose	:=FALSE;
				iVPolish.IO.doRelayLClose	:=FALSE;
				sVPolishState:=enOPEN;
			END_IF;

		enOPEN:
			iVPolish.IO.doRelayLOpen :=TRUE;
			iVPolish.IO.doRelayROpen :=TRUE;
			IF (iVPolish.IO.aiVPLForceF <= 5.0) AND (iVPolish.IO.aiVPRForceF <= 5.0 ) THEN
				iVPolish.IO.doRelayLClose :=FALSE;
				iVPolish.IO.doRelayRClose :=FALSE;
				sVPolishState:=enCLOSE;
			END_IF;
			//	(iVPolish.IO.aiVBLForceS >120 AND iVPolish.IO.aiVBRForceS >120)

		enCLOSE:
			iVPolish.IO.doRelayRClose:=TRUE;
			iVPolish.IO.doRelayLClose:=TRUE;

			IF (iVPolish.IO.aiVPLForceS > 120) AND (iVPolish.IO.aiVPRForceS > 120) THEN
				sVPolishState:=enOPERATION;
			END_IF;

		enOPERATION:
			iVPolish.IO.doRelayRClose:=FALSE;
			iVPolish.IO.doRelayLClose:=FALSE;
			IF (iVPolish.IO.aiVPLForceS =0 AND iVPolish.IO.aiVPRForceS =0) THEN
				sVPolishState:=enSTART;
			END_IF;

		enERROR:
			iVPolish.IO.doRelayLClose:=FALSE;
			iVPolish.IO.doRelayRClose:=FALSE;
			iVPolish.IO.doRelayRClose:=FALSE;
			iVPolish.IO.doRelayLClose:=FALSE;

			IF iVPolish.Cmd.ErrorReset=TRUE THEN
				iVPolish.Status.Error:=FALSE;
				iVPolish.Cmd.EStop	 :=FALSE;
				iVPolish.Cmd.ErrorReset:=FALSE;
				sVPolishState:=enSTART;
			END_IF;

	END_CASE;
END_PROGRAM

PROGRAM _EXIT
	(* Insert code here *)

END_PROGRAM
```

### Program Logical/Source/OptWax/WaxCtrl (IEC)

#### Main.st - Init, cyclic, exit code
```iecst
PROGRAM _INIT
	(* Insert code here *)

END_PROGRAM

PROGRAM _CYCLIC
	(* Insert code here *)
	WaxAlarm;
	IF iWax.Status.Error=TRUE THEN
		iWaxState:=enERROR;
	END_IF;
	CASE iWaxState OF

		enWAIT:

			iWax.Cmd.WaxRefill:= TRUE ;
			iWax.IO.doRealyWaxPump:=FALSE;
			iWax.IO.doValveWax:=FALSE;
			iWax.Status.PumpOn:=FALSE;
			iWax.Status.ValveOpen:=FALSE;
			iWax.Status.Running:=FALSE;

			IF iWax.Cmd.Start=TRUE THEN
				iWax.Cmd.WaxRefill	:= FALSE ;
				iWaxState:=enWAXON;
				iWax.Status.Running:=TRUE;
			END_IF;

		enWAXON:
			iWax.IO.doRealyWaxPump:=TRUE;
			iWax.IO.doValveWax:=TRUE;
			iWax.Status.PumpOn:=TRUE;
			iWax.Status.ValveOpen:=TRUE;

			IF iWax.IO.doRealyWaxPump=FALSE THEN
				iWaxState:=enWAIT;
			END_IF;

		enERROR:
			iWax.IO.doRealyWaxPump:=FALSE;
			iWax.IO.doValveWax:=FALSE;
			iWax.Status.PumpOn:=FALSE;
			iWax.Status.ValveOpen:=FALSE;
			iWax.Status.Running:=FALSE;
			IF iWax.Cmd.ErrorReset = TRUE THEN
				iWax.Cmd.ErrorReset:=FALSE;
				iWax.Cmd.EStop:=FALSE;
				iWax.Status.Error:=FALSE;
				iWaxState:=enWAIT;
			END_IF;

	END_CASE;
END_PROGRAM

PROGRAM _EXIT
	(* Insert code here *)

END_PROGRAM
```

#### Types.typ - Local data types
```iecst
TYPE
	sStep :
		(
		enWAIT,
		enWAXON,
		enERROR
		);
END_TYPE
```

#### Variables.var - Local variables
```iecst
VAR
	iWax : WaxCtrl_typ; (*main control*)
	iWaxState : sStep; (*enum of wax*)
END_VAR
```

#### WaxAlarm.st
```iecst
ACTION WaxAlarm:

	IF iWax.Cmd.EStop=TRUE THEN
		MpAlarmXSet(gAlarmXCore,'EStopHWax');
		IF MpAlarmXCheckReaction(gAlarmXCore, 'EStopErr') THEN
			iWax.Status.Error:= TRUE ;
		END_IF
	ELSE
		MpAlarmXReset(gAlarmXCore,'EStopHWax');
	END_IF;

END_ACTION
```

### WaxCtrl.typ
```iecst
TYPE
	WaxCmd_typ : 	STRUCT
		Start : BOOL;
		EStop : BOOL;
		Stop : BOOL;
		ErrorReset : BOOL;
		WaxRefill : BOOL;
	END_STRUCT;
	New_Datatype : 	STRUCT
	END_STRUCT;
	WaxCtrl_typ : 	STRUCT
		Cmd : WaxCmd_typ;
		IO : WaxIOs_typ;
		Par : WaxParam_typ;
		Status : WaxStatus_typ;
		WaxRefill : BOOL;
	END_STRUCT;
	WaxIOs_typ : 	STRUCT
		doValveWax : BOOL;
		doRealyWaxPump : BOOL;
		doRefillWax : BOOL;
		WaxRefill : BOOL;
	END_STRUCT;
	WaxParam_typ : 	STRUCT
		New_Member : USINT;
	END_STRUCT;
	WaxStatus_typ : 	STRUCT
		Running : BOOL;
		Error : BOOL;
		PumpOn : BOOL;
		ValveOpen : BOOL;
	END_STRUCT;
END_TYPE
```

### Program Logical/Source/Drying/DryHCtrl (IEC)

#### Main.st - Init, cyclic, exit code
```iecst
PROGRAM _INIT
	(* Insert code here *)

END_PROGRAM

PROGRAM _CYCLIC
	(* Insert code here *)
	DryAlarm;
	IF iDry.Status.Error=TRUE THEN
		sDryState:=enERROR;
	END_IF;

	CASE sDryState OF

		enWAIT:
			IF iDry.Cmd.Start = TRUE THEN
				sDryState		:= enSTART;
			END_IF;

		enSTART:
			IF (iDry.IO.diSens1Dry1 = FALSE) AND (iDry.IO.diSens1Dry2 = FALSE) AND (iDry.IO.diSens1Dry3 = FALSE) AND (iDry.IO.diSens1Dry4 = FALSE) THEN
				iDry.IO.doRelayHD1Lower	:= TRUE;
				iDry.IO.doRelayHD1Lift	:= FALSE;
				iDry.IO.doRelayVDHeater	:=TRUE;
				iDry.IO.doRelayVDVent	:=TRUE;
				iDry.IO.doRelayHD1Vent	:= TRUE;
				iDry.IO.doRelayHD1Heater:= TRUE;
			END_IF;

			IF (iDry.IO.diSens1Dry1 = TRUE) AND (iDry.IO.diSens1Dry2 = FALSE) AND (iDry.IO.diSens1Dry3 = FALSE) AND (iDry.IO.diSens1Dry4 = FALSE) THEN
				iDry.IO.doRelayHD1Lower		:= FALSE;
				iDry.IO.doRelayHD1Lift		:= FALSE;
				sDryState					:= enOPERATION;
			END_IF;
		enOPERATION:
			IF (iDry.IO.diSens1Dry1 = TRUE) AND (iDry.IO.diSens1Dry2 = FALSE) AND (iDry.IO.diSens1Dry3 = FALSE) AND (iDry.IO.diSens1Dry4 = FALSE) THEN
				iDry.IO.doRelayHD1Lower	:= FALSE;
				iDry.IO.doRelayHD1Lift	:= FALSE;
			END_IF;

			IF (iDry.IO.diSens1Dry1 = TRUE) AND (iDry.IO.diSens1Dry2 = TRUE) AND (iDry.IO.diSens1Dry3 = TRUE) AND (iDry.IO.diSens1Dry4 = FALSE) THEN
				iDry.IO.doRelayHD1Lower	:= FALSE;
				iDry.IO.doRelayHD1Lift	:= TRUE;
			END_IF;

			IF (iDry.IO.diSens1Dry1 = TRUE) AND (iDry.IO.diSens1Dry2 = TRUE) AND (iDry.IO.diSens1Dry3 = FALSE) AND (iDry.IO.diSens1Dry4 = FALSE) THEN
				iDry.IO.doRelayHD1Lower	:= FALSE;
				iDry.IO.doRelayHD1Lift	:= TRUE;
			END_IF;

			IF (iDry.IO.diSens1Dry1 = FALSE) AND (iDry.IO.diSens1Dry2 = FALSE) AND (iDry.IO.diSens1Dry3 = TRUE) AND (iDry.IO.diSens1Dry4 = FALSE) THEN
				iDry.IO.doRelayHD1Lower	:= TRUE;
				iDry.IO.doRelayHD1Lift	:= FALSE;
			END_IF;

			IF (iDry.IO.diSens1Dry1 = FALSE) AND (iDry.IO.diSens1Dry2 = FALSE) AND (iDry.IO.diSens1Dry3 = TRUE) AND (iDry.IO.diSens1Dry4 = TRUE) THEN
				iDry.IO.doRelayHD1Lower	:= FALSE;
				iDry.IO.doRelayHD1Lift	:= FALSE;
			END_IF;

			IF (iDry.IO.diSens1Dry1 = FALSE) AND (iDry.IO.diSens1Dry2 = FALSE) AND (iDry.IO.diSens1Dry3 = FALSE) AND (iDry.IO.diSens1Dry4 = FALSE) THEN
				iDry.IO.doRelayHD1Lower	:= FALSE;
				iDry.IO.doRelayHD1Lift	:= FALSE;
				iDry.IO.doRelayHD1Vent	:= FALSE;
				iDry.IO.doRelayHD1Heater:= FALSE;
				iDry.IO.doRelayHD1Vent	:= FALSE;
				iDry.IO.doRelayHD1Heater:= FALSE;
//				iDry.Cmd.Start		:= FALSE;
//				sDryState				:= enWAIT;
			END_IF;

		enERROR:
			iDry.IO.doRelayHD1Lower	:= FALSE;
			iDry.IO.doRelayHD1Lift	:= FALSE;
			iDry.IO.doRelayHD1Vent	:= FALSE;
			iDry.IO.doRelayHD1Heater:= FALSE;
			iDry.IO.doRelayHD1Vent	:= FALSE;
			iDry.IO.doRelayHD1Heater:= FALSE;
			IF iDry.Cmd.ErrorReset=TRUE THEN
				iDry.Cmd.ErrorReset	:=FALSE;
				iDry.Cmd.EStop		:=FALSE;
				iDry.Status.Error	:=FALSE;
				sDryState:=enWAIT;
			END_IF;
	END_CASE;

END_PROGRAM

PROGRAM _EXIT
	(* Insert code here *)

END_PROGRAM
```

#### Variables.var - Local variables
```iecst
VAR
	sDryState : sStep_enum; (*dry enum*)
	iDry : DryCtrl_typ; (*main control*)
END_VAR
```

#### DryAlarm.st
```iecst
ACTION DryAlarm:
	IF iDry.Cmd.EStop=TRUE THEN
		MpAlarmXSet(gAlarmXCore,'EStopDry');
		IF MpAlarmXCheckReaction(gAlarmXCore, 'EStopErr') THEN
			iDry.Status.Error:= TRUE ;
		END_IF
	ELSE
		MpAlarmXReset(gAlarmXCore,'EStopDry');
	END_IF;
END_ACTION
```

### Program Logical/Source/Drying/DryH2Ctrl (IEC)

#### Types.typ
```iecst
TYPE
	sStep_enum :
		(
		enWAIT,
		enSTART,
		enOPEN,
		enOPERATION,
		enCLOSE,
		enERROR
		);
END_TYPE
```

#### Variables.var
```iecst
VAR
	sDryState : sStep_enum; (*dry enum*)
	iDry2 : DryCtrl_typ; (*main control*)
	sDryState2 : sStep_enum; (*enumeration of drystate*)
END_VAR
```

#### Main.st
```iecst
PROGRAM _INIT
	(* Insert code here *)

END_PROGRAM

PROGRAM _CYCLIC
	(* Insert code here *)

	CASE sDryState2 OF

		enWAIT:
			IF iDry2.Cmd.Start = TRUE THEN
				sDryState2		:= enSTART;
			END_IF;

		enSTART:
			IF (iDry2.IO.diSens2Dry1 = FALSE) AND (iDry2.IO.diSens2Dry2 = FALSE) AND (iDry2.IO.diSens2Dry3 = FALSE) AND (iDry2.IO.diSens2Dry4 = FALSE) THEN
				iDry2.IO.doRelayHD2Lower	:= TRUE;
				iDry2.IO.doRelayHD2Lift	:= FALSE;
				iDry2.IO.doRelayHD2Vent	:= TRUE;
				iDry2.IO.doRelayHD2Heater:= TRUE;
			END_IF;
			IF (iDry2.IO.diSens2Dry1 = TRUE) AND (iDry2.IO.diSens2Dry2 = FALSE) AND (iDry2.IO.diSens2Dry3 = FALSE) AND (iDry2.IO.diSens2Dry4 = FALSE) THEN
				iDry2.IO.doRelayHD2Lower	:= FALSE;
				iDry2.IO.doRelayHD2Lift		:= FALSE;
				sDryState2					:= enOPERATION;
			END_IF;
		enOPERATION:
			IF (iDry2.IO.diSens2Dry1 = TRUE) AND (iDry2.IO.diSens2Dry2 = FALSE) AND (iDry2.IO.diSens2Dry3 = FALSE) AND (iDry2.IO.diSens2Dry4 = FALSE) THEN
				iDry2.IO.doRelayHD2Lower	:= FALSE;
				iDry2.IO.doRelayHD2Lift	:= FALSE;
			END_IF;
			IF (iDry2.IO.diSens2Dry1 = TRUE) AND (iDry2.IO.diSens2Dry2 = TRUE) AND (iDry2.IO.diSens2Dry3 = TRUE) AND (iDry2.IO.diSens2Dry4 = FALSE) THEN
				iDry2.IO.doRelayHD2Lower	:= FALSE;
				iDry2.IO.doRelayHD2Lift	:= TRUE;
			END_IF;
			IF (iDry2.IO.diSens2Dry1 = TRUE) AND (iDry2.IO.diSens2Dry2 = TRUE) AND (iDry2.IO.diSens2Dry3 = FALSE) AND (iDry2.IO.diSens2Dry4 = FALSE) THEN
				iDry2.IO.doRelayHD2Lower	:= FALSE;
				iDry2.IO.doRelayHD2Lift	:= TRUE;
			END_IF;
			IF (iDry2.IO.diSens2Dry1 = FALSE) AND (iDry2.IO.diSens2Dry2 = FALSE) AND (iDry2.IO.diSens2Dry3 = TRUE) AND (iDry2.IO.diSens2Dry4 = FALSE) THEN
				iDry2.IO.doRelayHD2Lower	:= TRUE;
				iDry2.IO.doRelayHD2Lift	:= FALSE;
			END_IF;
			IF (iDry2.IO.diSens2Dry1 = FALSE) AND (iDry2.IO.diSens2Dry2 = FALSE) AND (iDry2.IO.diSens2Dry3 = TRUE) AND (iDry2.IO.diSens2Dry4 = TRUE) THEN
				iDry2.IO.doRelayHD2Lower	:= FALSE;
				iDry2.IO.doRelayHD2Lift	:= FALSE;
			END_IF;
			IF (iDry2.IO.diSens2Dry1 = FALSE) AND (iDry2.IO.diSens2Dry2 = FALSE) AND (iDry2.IO.diSens2Dry3 = FALSE) AND (iDry2.IO.diSens2Dry4 = FALSE) THEN
				iDry2.IO.doRelayHD2Lower	:= FALSE;
				iDry2.IO.doRelayHD2Lift	:= FALSE;
				iDry2.IO.doRelayVDHeater	:=FALSE;
				iDry2.IO.doRelayVDVent	:=FALSE;
//				iDry2.Cmd.Start		:= FALSE;
//				sDryState2				:= enWAIT;
			END_IF;

		enERROR:
			iDry2.IO.doRelayHD2Lower	:= FALSE;
			iDry2.IO.doRelayHD2Lift	:= FALSE;
			iDry2.IO.doRelayVDHeater	:=FALSE;
			iDry2.IO.doRelayVDVent	:=FALSE;
			iDry2.Cmd.Start			:= FALSE;
			IF iDry2.Cmd.ErrorReset=TRUE THEN
				iDry2.Status.Error	:=FALSE;
				sDryState:=enWAIT;
			END_IF;

	END_CASE;

END_PROGRAM

PROGRAM _EXIT
	(* Insert code here *)

END_PROGRAM
```

### DryCtrl.typ
```iecst
TYPE
	DryCmd_typ : 	STRUCT
		Start : BOOL;
		EStop : BOOL;
		Stop : BOOL;
		ErrorReset : BOOL;
	END_STRUCT;
	DryCtrl_typ : 	STRUCT
		Cmd : DryCmd_typ;
		IO : DryIOs_typ;
		Par : DryParam_typ;
		Status : DryStatus_typ;
	END_STRUCT;
	DryIOs_typ : 	STRUCT
		diSens1Dry1 : BOOL;
		diSens1Dry2 : BOOL;
		diSens1Dry3 : BOOL;
		diSens1Dry4 : BOOL;
		diSens2Dry2 : BOOL;
		diSens2Dry3 : BOOL;
		diSens2Dry4 : BOOL;
		diSens2Dry1 : BOOL;
		doRelayHD1Lower : BOOL;
		doRelayHD1Vent : BOOL;
		doRelayHD1Heater : BOOL;
		doRelayVDVent : BOOL;
		doRelayVDHeater : BOOL;
		doRelayHD1Lift : BOOL;
		doRelayHD2Lower : BOOL;
		doRelayHD2Vent : BOOL;
		doRelayHD2Heater : BOOL;
		doRelayHD2Lift : BOOL;
	END_STRUCT;
	DryParam_typ : 	STRUCT
		New_Member : USINT;
	END_STRUCT;
	DryStatus_typ : 	STRUCT
		Running : BOOL;
		Error : BOOL;
	END_STRUCT;
END_TYPE
```

### Program Logical/Source/CarExit/CarExit (IEC)

#### Main.st - Init, cyclic, exit code
```iecst
PROGRAM _INIT

END_PROGRAM

PROGRAM _CYCLIC
	ExitAlarm;
	IF iExit.Status.Error=TRUE THEN
		sExitState:=enERROR;
	END_IF;
	CASE sExitState OF

		enWAIT:

			IF iExit.Cmd.Start=TRUE  THEN
				sExitState:=enSTART;
			END_IF;

		enSTART:
			iExit.IO.doRelayLiftDoor:=TRUE;

			iExit.Status.LiftingDoor:=TRUE;

		enOPERATION:
			iExit.IO.doRelayLowerdDoor:=TRUE;

			iExit.Status.LowringDoor:=TRUE;
		enERROR:

			iExit.IO.doGreenLight	:=FALSE;
			iExit.IO.doOrangeLight	:=FALSE;
			iExit.IO.doRedLight		:=FALSE;
			iExit.IO.doRelayLiftDoor:=FALSE;
			iExit.Status.LiftingDoor:=FALSE;
			iExit.Status.LowringDoor:=FALSE;
			IF iExit.Cmd.ErrorReset = TRUE THEN
				iExit.Cmd.ErrorReset:=FALSE;
				iExit.Cmd.EStop		:=FALSE;
				iExit.Status.Error	:=FALSE;
				sExitState			:=enWAIT;
			END_IF;
	END_CASE;
END_PROGRAM

PROGRAM _EXIT

				END_PROGRAM
```

#### Types.typ - Local data types
```iecst
TYPE
	sStep_enum :
		(
		enWAIT,
		enSTART,
		enOPERATION,
		enERROR
		);
END_TYPE
```

#### Variables.var - Local variables
```iecst
VAR
	iExit : CarExitCtrl_typ;
	sExitState : sStep_enum;
END_VAR
```

#### ExitAlarm.st
```iecst
ACTION ExitAlarm:
	IF iExit.Cmd.EStop=TRUE THEN
		MpAlarmXSet(gAlarmXCore,'EStopExit');
		IF MpAlarmXCheckReaction(gAlarmXCore, 'EStopErr') THEN
			iExit.Status.Error:= TRUE ;
		END_IF
	ELSE
		MpAlarmXReset(gAlarmXCore,'EStopExit');
	END_IF;
END_ACTION
```

### CarExit.typ
```iecst
TYPE
	CarExitCmd_typ : 	STRUCT
		Start : BOOL;
		EStop : BOOL;
		Stop : BOOL;
		ErrorReset : BOOL;
	END_STRUCT;
	CarExitCtrl_typ : 	STRUCT
		Cmd : CarExitCmd_typ;
		IO : CarExitIOs_typ;
		Par : CarExitParam_typ;
		Status : CarExitStatus_typ;
	END_STRUCT;
	CarExitIOs_typ : 	STRUCT
		doGreenLight : BOOL;
		doRelayLowerdDoor : BOOL;
		doRelayLiftDoor : BOOL;
		doRedLight : BOOL;
		doOrangeLight : BOOL;
	END_STRUCT;
	CarExitParam_typ : 	STRUCT
		New_Member : USINT;
	END_STRUCT;
	CarExitStatus_typ : 	STRUCT
		Running : BOOL;
		Error : BOOL;
		LiftingDoor : BOOL;
		LowringDoor : BOOL;
	END_STRUCT;
END_TYPE
```

### Program Logical/Source/Infrastructure/AlarmCtrl/AlarmCtrl

#### Variables.var
```iecst
VAR
	iFb_AlarmX : MpAlarmXCore;
	iFb_AlarmUI : MpAlarmXListUI;
	UIConnectCore : MpAlarmXListUIConnectType;
END_VAR
```

#### Main.st
```iecst
PROGRAM _INIT
	(* Insert code here *)

END_PROGRAM

PROGRAM _CYCLIC

	// alarmx on
	iFb_AlarmX.Enable:=TRUE;
	iFb_AlarmX.MpLink:=ADR(gAlarmXCore);

	iFb_AlarmUI.Enable:=TRUE;
	iFb_AlarmUI.MpLink:=ADR(gAlarmXCore);
	iFb_AlarmUI.UIConnect:=ADR(UIConnectCore);

	iFb_AlarmX();
	iFb_AlarmUI();
END_PROGRAM

PROGRAM _EXIT
	(* Insert code here *)

	iFb_AlarmUI.Enable:=FALSE;
	iFb_AlarmX.Enable:=FALSE;
	iFb_AlarmX();
	iFb_AlarmUI();
END_PROGRAM
```

### Program Logical/Source/Infrastructure/DataCtrl/DataCtrl (IEC)

#### Variables.var
```iecst
VAR
	iFb_DataRecorder : MpDataRecorder;
	iFb_DataParMode1 : MpDataRegPar;
	iFb_DataParMode2 : MpDataRegPar;
	iFb_DataParMode3 : MpDataRegPar;
	iFb_DataParMode4 : MpDataRegPar;
END_VAR
```

#### Main.st
```iecst
PROGRAM _INIT
	(* Insert code here *)
	gMi_Mode1 ;
	gMi_Mode2 ;
	gMi_Mode3 ;
	gMi_Mode4 ;
END_PROGRAM

PROGRAM _CYCLIC
	(* Insert code here *)
	//Data Recorder for two parameter of Feed Change
	iFb_DataRecorder.Enable := TRUE ;
	iFb_DataRecorder.DeviceName := ADR('USER') ;
	iFb_DataRecorder.MpLink := ADR(gDataRecorder);
	iFb_DataRecorder.RecordMode := mpDATA_RECORD_MODE_VALUE ;

	iFb_DataParMode1.Enable := TRUE ;
	iFb_DataParMode1.MpLink := ADR(gDataRecorder);
	iFb_DataParMode1.PVName := ADR ('gMi_Mode1') ;

	iFb_DataParMode2.Enable := TRUE ;
	iFb_DataParMode2.MpLink := ADR(gDataRecorder);
	iFb_DataParMode2.PVName := ADR ('gMi_Mode2') ;
	iFb_DataParMode3.Enable := TRUE ;
	iFb_DataParMode3.MpLink := ADR(gDataRecorder);
	iFb_DataParMode3.PVName := ADR ('gMi_Mode3') ;
	iFb_DataParMode4.Enable := TRUE ;
	iFb_DataParMode4.MpLink := ADR(gDataRecorder);
	iFb_DataParMode4.PVName := ADR ('gMi_Mode4') ;
	IF iFb_DataRecorder.Active = TRUE AND iFb_DataRecorder.StatusID = 0 THEN
		iFb_DataRecorder.Record := TRUE;
	END_IF
	iFb_DataParMode1 ();
	iFb_DataParMode2 ();
	iFb_DataParMode3 () ;
	iFb_DataParMode4 () ;
	iFb_DataRecorder();
	END_PROGRAM

PROGRAM _EXIT
	(* Insert code here *)
	iFb_DataRecorder.Enable := FALSE ;
	iFb_DataRecorder();
END_PROGRAM
```

- Visualisation Logical/Source/VisuCtrl (not shown)

### Program Logical/Source/Auxillary/Auxillary (IEC)

#### Variables.var
```iecst
VAR
	iAuxillary : Auxillary_typ;
END_VAR
```

#### Main.st
```iecst
PROGRAM _INIT
	(* Insert code here *)

END_PROGRAM

PROGRAM _CYCLIC
	(* Insert code here *)
	iAuxillary;
END_PROGRAM

PROGRAM _EXIT
	(* Insert code here *)

END_PROGRAM
```

### Types.typ
```iecst
TYPE
	Auxillary_typ : 	STRUCT
		doRelayConv : BOOL;
	END_STRUCT;
END_TYPE
```

### Program Logical/Source/HPolishp/HPolish (IEC)
